// TIA Portal V20 export
// export: Created 2026-04-23T02:21:41.3399534Z, ExportSetting None, DisplayName Totally Integrated Automation Portal, DisplayVersion V20 Update 4, DisplayName TIA Portal Openness, DisplayVersion V20 Update 4, DisplayName TIA Portal Version Control Interface, DisplayVersion V20 Update 4, DisplayName SINAMICS Startdrive Advanced, DisplayVersion V20 SP1 Update 2, DisplayName SINAMICS Startdrive G110M, G120, G120C, G120D, G120P, G115D, DisplayVersion V20 SP1 Update 2, DisplayName SINAMICS Startdrive G130, G150, S120, S150, SINAMICS MV, G220, S200, S210, DisplayVersion V20 SP1 Update 2, DisplayName STEP 7 Professional, DisplayVersion V20 Update 4, DisplayName STEP 7 Safety, DisplayVersion V20 Update 2, DisplayName WinCC Basic/Comfort/Advanced, DisplayVersion V20 Update 4, DisplayName SIMATIC Visualization Architect, DisplayVersion V20 Update 4, DisplayName WinCC Unified, DisplayVersion V20 Update 4, DisplayName SIMATIC Visualization Architect, DisplayVersion V20 Update 4
FUNCTION_BLOCK "LSicar_KistlerPress"   // FB2, LAD
{ S7_Optimized_Access := 'TRUE' }
// stored: MemoryReserve 100, SetENOAutomatically false
   VAR_INPUT
      plantidentifier { ExternalAccessible := 'False'; ExternalVisible := 'False'; ExternalWritable := 'False'} : WString[24];   // Plant/cell identifier string (max 24 chars). Embedded in all ProDiag alarm messages via the @5%s@ placeholder. Set to a unique name per press instance, e.g. KP_ST110_PRS1.
      CarrierID { ExternalAccessible := 'False'; ExternalVisible := 'False'; ExternalWritable := 'False'} : WString[9];   // Carrier or pallet ID (max 9 chars). Passed to the Kistler SmartClient to correlate measurement results with the workpiece carrier for traceability.
      mpSerialNumber { ExternalAccessible := 'False'; ExternalVisible := 'False'; ExternalWritable := 'False'} : String[24];   // Expected workpiece serial number (max 24 chars). Compared against the serial reported by the Kistler device each cycle. A mismatch sets stateAlarm.serialnumbermismatch and blocks sequence start.
      additionaAlarmText { ExternalAccessible := 'False'; ExternalVisible := 'False'; ExternalWritable := 'False'} : WString[15];   // Additional context text (max 15 chars) appended to alarm messages. Use for extra identification, e.g. tool number or station sub-ID.
      tecUnitNumber { ExternalAccessible := 'False'; ExternalVisible := 'False'; ExternalWritable := 'False'} : Int;   // Technical unit number for this press instance. Used for HMI interface routing and identification in multi-press installations.
      enableBlock { ExternalAccessible := 'False'; ExternalVisible := 'False'; ExternalWritable := 'False'} : Bool := TRUE;   // Master block enable. TRUE = block logic active and outputs driven. FALSE = all drive outputs de-energised and alarms suppressed. Default TRUE.
      HardwareOK { ExternalAccessible := 'False'; ExternalVisible := 'False'; ExternalWritable := 'False'} : Bool := TRUE;   // Fieldbus and drive hardware health input. FALSE triggers stateAlarm.hardwareNOK and inhibits all motion commands. Connect to PROFINET device diagnostic or drive ready signal. Default TRUE.
      SafetyOK { ExternalAccessible := 'False'; ExternalVisible := 'False'; ExternalWritable := 'False'} : Bool := TRUE;   // Safety circuit status. FALSE gates all motion commands, de-energises the drive enable, and sets stateAlarm.safetyNOK. Must be TRUE before any press movement is permitted. Default TRUE.
      servoNotInstalled { ExternalAccessible := 'False'; ExternalVisible := 'False'; ExternalWritable := 'False'} : Bool;   // Set TRUE when the servo drive is physically absent (spare station). Bypasses drive-enable and drive-fault alarms and allows the block to run in passthrough mode without a physical axis.
      hardwareID1 { ExternalAccessible := 'False'; ExternalVisible := 'False'; ExternalWritable := 'False'} : HW_IO;   // TIA hardware identifier (HW_IO) for the primary Kistler PROFINET device. Used as LADDR in DPRD_DAT to read the 200-byte cyclic receive telegram each scan.
      hardwareID2 { ExternalAccessible := 'False'; ExternalVisible := 'False'; ExternalWritable := 'False'} : HW_IO;   // TIA hardware identifier (HW_IO) for the secondary Kistler PROFINET device. Used as LADDR in DPWR_DAT to write the transmit telegram to the device.
      smartClientIPAddress { ExternalAccessible := 'False'; ExternalVisible := 'False'; ExternalWritable := 'False'} : String[20];   // IP address string of the Kistler SmartClient application (max 20 chars). Stored for reference and remote configuration. Set to the network address of the Kistler PC running SmartClient.
      mpNumber { ExternalAccessible := 'False'; ExternalVisible := 'False'; ExternalWritable := 'False'} : Byte;   // Measurement program (MP) number to load on the Kistler device. Sent via the fieldbus transmit telegram. Valid range and program definitions are configured on the Kistler SmartClient.
      cfgAdd { ExternalAccessible := 'False'; ExternalVisible := 'False'; ExternalWritable := 'False'} : Byte;   // Starting byte offset in the Kistler fieldbus configuration area. Combined with CfgLentgh to define the read/write window for the configuration data telegram exchange.
      CfgLentgh { ExternalAccessible := 'False'; ExternalVisible := 'False'; ExternalWritable := 'False'} : Byte;   // Length in bytes of the Kistler configuration telegram block. Determines how many bytes are transferred during each configuration read or write operation.
      SelectPageNumber { ExternalAccessible := 'False'; ExternalVisible := 'False'; ExternalWritable := 'False'} : Byte;   // Display page number to activate on the Kistler operator panel or SmartClient HMI. Sent in the transmit telegram each scan.
      selectSequence { ExternalAccessible := 'False'; ExternalVisible := 'False'; ExternalWritable := 'False'} : Byte;   // Sequence profile number to activate on the Kistler device. Sent via the fieldbus transmit telegram to select which measurement sequence to run.
      extStopRequest { ExternalAccessible := 'False'; ExternalVisible := 'False'; ExternalWritable := 'False'} : Bool;   // External stop request from upstream logic (e.g. part-not-present or conveyor fault). Rising edge halts the running sequence gracefully and sets sequenceStopped. Timeout monitored by timeExtStop.
      strobeEnable { ExternalAccessible := 'False'; ExternalVisible := 'False'; ExternalWritable := 'False'} : Bool;   // Gate for the automatic data-strobe pulse. TRUE allows the strobe command to be sent to the Kistler device during a running sequence to trigger data capture.
      startTL { ExternalAccessible := 'False'; ExternalVisible := 'False'; ExternalWritable := 'False'} : Bool;   // Rising edge initiates the teach-learn or reference-position calibration cycle on the Kistler axis. Hold TRUE until the TL cycle is confirmed complete.
      autoRunSequence { ExternalAccessible := 'False'; ExternalVisible := 'False'; ExternalWritable := 'False'} : Bool := FALSE;   // When TRUE the block automatically triggers the measurement sequence on each new cycle trigger. When FALSE the sequence must be started manually via HMI. Default FALSE.
      autoHomePosition { ExternalAccessible := 'False'; ExternalVisible := 'False'; ExternalWritable := 'False'} : Bool;   // When TRUE the axis automatically returns to home position after each sequence completes normally. Disable for processes that require the axis to hold position after pressing.
      autoDriveToReferencePosition { ExternalAccessible := 'False'; ExternalVisible := 'False'; ExternalWritable := 'False'} : Bool;   // When TRUE the axis automatically drives to the reference/calibration position during block initialisation or after a reset. Used for absolute position referencing at startup.
      JogFwd { ExternalAccessible := 'False'; ExternalVisible := 'False'; ExternalWritable := 'False'} : Bool;   // Jog press forward (downward, pressing direction). Drive moves while signal is TRUE. Only active in manual or setup mode. Rate limited by jog speed in parameters.
      JogNeq { ExternalAccessible := 'False'; ExternalVisible := 'False'; ExternalWritable := 'False'} : Bool;   // Jog press negative/backward (upward, retract direction). Drive moves while signal is TRUE. Only active in manual or setup mode.
      continuewait { ExternalAccessible := 'False'; ExternalVisible := 'False'; ExternalWritable := 'False'} : Bool;   // Rising edge clears the waitContinue pause state and resumes sequence execution. Used for operator-confirmation steps in semi-automatic cycles or fault-recovery sequences.
      SequenceEndReset { ExternalAccessible := 'False'; ExternalVisible := 'False'; ExternalWritable := 'False'} : Bool;   // Rising edge resets the Sequenceend, sequenceStopped, and internal sequence-complete flags, clearing the end-of-cycle indication and allowing a new cycle to be triggered.
      enableRunSequence { ExternalAccessible := 'False'; ExternalVisible := 'False'; ExternalWritable := 'False'} : Bool := TRUE;   // Enable gate for sequence execution. FALSE prevents the measurement sequence from starting even if autoRunSequence is TRUE or a manual start is requested. Default TRUE.
      enablehomePos { ExternalAccessible := 'False'; ExternalVisible := 'False'; ExternalWritable := 'False'} : Bool := TRUE;   // Enable gate for home-position return. FALSE prevents the axis from driving to home position even when autoHomePosition is TRUE. Default TRUE.
      externalAlarm { ExternalAccessible := 'False'; ExternalVisible := 'False'; ExternalWritable := 'False'} : Bool;   // External fault injection from another block or interlock. When TRUE, sets stateAlarm.alarm and contributes to GeneralAlarm. Allows upstream faults to be reflected through the Kistler block.
      runWithoutEnable { ExternalAccessible := 'False'; ExternalVisible := 'False'; ExternalWritable := 'False'} : Bool;   // Bypass flag for the opmode enable check. When TRUE the block runs in automatic mode even if the opmode enable signal is not active. Use for commissioning only.
      hideAlarmAll { ExternalAccessible := 'False'; ExternalVisible := 'False'; ExternalWritable := 'False'} : Bool;   // Global alarm suppression. When TRUE all ProDiag alarm messages are suppressed. Does not clear active faults, only prevents message annunciation. Typically driven by a plant-level inhibit.
      hideAlarmMask { ExternalAccessible := 'False'; ExternalVisible := 'False'; ExternalWritable := 'False'} : DWord;   // 32-bit individual alarm suppression mask. Each bit maps to one stateAlarm bit (bit 0 = spare0, bit 1 = hardwareNOK, etc.). Set a bit TRUE to suppress that alarm channel without affecting others.
      OpModeUserInterfaceOut { ExternalAccessible := 'False'; ExternalVisible := 'False'; ExternalWritable := 'False'} : "LSicar_typeOpmodeOut";   // Operating mode data from SYSTEM_DB.OPmode[N].User_Interface_OUT. Contains automaticActive, manualActive, singleStepActive flags and operator preselect requests used to drive mode-selection logic.
      timeOperation { ExternalAccessible := 'False'; ExternalVisible := 'False'; ExternalWritable := 'False'} : Time;   // Maximum allowed duration for a press operation cycle (IEC Time). If the sequence does not complete within this time, stateAlarm.timerMonitorRunSequence is set and the cycle is aborted.
      timeExtStop { ExternalAccessible := 'False'; ExternalVisible := 'False'; ExternalWritable := 'False'} : Time;   // Maximum time allowed for the extStopRequest signal to clear after it rises. If the signal remains TRUE beyond this time, a timeout fault is latched in stateAlarm.
      parameters { ExternalAccessible := 'False'; ExternalVisible := 'False'; ExternalWritable := 'False'} : "LDrive_typeKistlerParameters";   // LDrive_typeKistlerParameters struct. Contains press axis travel limits, force window limits, jog speed, sequence timing parameters, and SmartClient configuration values.
   END_VAR
   VAR_OUTPUT
      GeneralAlarm { ExternalAccessible := 'False'; ExternalVisible := 'False'; ExternalWritable := 'False'} : Bool;   // TRUE when any active unmasked fault condition exists. Drives ProDiag supervision alarm output. Must be FALSE for the ready output to be TRUE.
      AutomaticActive { ExternalAccessible := 'False'; ExternalVisible := 'False'; ExternalWritable := 'False'} : Bool;   // TRUE when the block is operating in automatic mode (opmode automatic active and enableBlock TRUE). Indicates the press is available for production cycles.
      okTotal { ExternalAccessible := 'False'; ExternalVisible := 'False'; ExternalWritable := 'False'} : Bool;   // Pulses TRUE for one scan when the Kistler device reports an OK result for the last completed measurement (all evaluation channels within defined limits).
      nokTotal { ExternalAccessible := 'False'; ExternalVisible := 'False'; ExternalWritable := 'False'} : Bool;   // Pulses TRUE for one scan when the Kistler device reports a NOK result (at least one evaluation channel outside its defined limit window).
      noPass { ExternalAccessible := 'False'; ExternalVisible := 'False'; ExternalWritable := 'False'} : Bool;   // TRUE when the Kistler evaluation reports a no-pass condition for the current measurement program. Distinct from NOK -- indicates an evaluation rule was not met.
      sequenceRunning { ExternalAccessible := 'False'; ExternalVisible := 'False'; ExternalWritable := 'False'} : Bool;   // TRUE while a measurement sequence is actively executing on the press axis. Falls FALSE when the sequence completes, is stopped, or a fault occurs.
      sequenceStopped { ExternalAccessible := 'False'; ExternalVisible := 'False'; ExternalWritable := 'False'} : Bool;   // TRUE after a sequence was interrupted by extStopRequest or a manual stop command. Remains TRUE until cleared by SequenceEndReset rising edge.
      Sequenceend { ExternalAccessible := 'False'; ExternalVisible := 'False'; ExternalWritable := 'False'} : Bool;   // Pulses TRUE for one scan when a sequence completes normally without fault. Cleared by SequenceEndReset rising edge or the start of a new cycle.
      homePos { ExternalAccessible := 'False'; ExternalVisible := 'False'; ExternalWritable := 'False'} : Bool;   // TRUE when the press axis is confirmed at the home/retracted position within the home-position tolerance window defined in parameters.
      referencePos { ExternalAccessible := 'False'; ExternalVisible := 'False'; ExternalWritable := 'False'} : Bool;   // TRUE when the press axis is confirmed at the reference/calibration position. Used to validate absolute position referencing after startup or reset.
      waitContinue { ExternalAccessible := 'False'; ExternalVisible := 'False'; ExternalWritable := 'False'} : Bool;   // TRUE when the block is paused at a wait-for-operator step in the sequence. Cleared by a rising edge on the continuewait input.
      ready { ExternalAccessible := 'False'; ExternalVisible := 'False'; ExternalWritable := 'False'} : Bool;   // TRUE when the block is fault-free, fully enabled, axis at home position, and ready to accept a new cycle trigger. The primary go/no-go signal for upstream sequence control.
      pvCurrentValueX { ExternalAccessible := 'False'; ExternalVisible := 'False'; ExternalWritable := 'False'} : Real;   // Live X-axis process value from the Kistler sensor, typically press position in mm. Scaled from the raw fieldbus data using engineering unit conversion in the Process Values Mapping network.
      pvCurrentValueY { ExternalAccessible := 'False'; ExternalVisible := 'False'; ExternalWritable := 'False'} : Real;   // Live Y-axis process value from the Kistler sensor, typically press force in kN. Scaled from the raw fieldbus data using engineering unit conversion in the Process Values Mapping network.
      pvCurveXminX { ExternalAccessible := 'False'; ExternalVisible := 'False'; ExternalWritable := 'False'} : Real;   // Lower X bound (position) of the active evaluation envelope window. Sourced from the current measurement program parameters on the Kistler device.
      pvCurveXmaxX { ExternalAccessible := 'False'; ExternalVisible := 'False'; ExternalWritable := 'False'} : Real;   // Upper X bound (position) of the active evaluation envelope window. Sourced from the current measurement program parameters on the Kistler device.
      pvCurveYminY { ExternalAccessible := 'False'; ExternalVisible := 'False'; ExternalWritable := 'False'} : Real;   // Lower Y bound (force) of the active evaluation envelope window. Sourced from the current measurement program parameters on the Kistler device.
      pvCurveYmaxY { ExternalAccessible := 'False'; ExternalVisible := 'False'; ExternalWritable := 'False'} : Real;   // Upper Y bound (force) of the active evaluation envelope window. Sourced from the current measurement program parameters on the Kistler device.
      customeProcessValues { ExternalAccessible := 'False'; ExternalVisible := 'False'; ExternalWritable := 'False'} : "LDrive_typeKistlerProcessValues";   // LDrive_typeKistlerProcessValues struct. Full result set from the Kistler evaluation: all channel measured values, individual pass/fail flags, peak force, peak position, and gradient data.
      displayeservoJogSpeed { ExternalAccessible := 'False'; ExternalVisible := 'False'; ExternalWritable := 'False'} : Real;   // Current servo jog speed as a percentage (0-100%). Calculated from the active jog speed parameter and displayed on the HMI for operator awareness during manual axis movement.
      standstill { ExternalAccessible := 'False'; ExternalVisible := 'False'; ExternalWritable := 'False'} : Bool;   // TRUE when the servo axis velocity is confirmed at zero by the drive. Safe condition for clamp operations or position checks that require the press to be stationary.
      MeasurementProgramEcho { ExternalAccessible := 'False'; ExternalVisible := 'False'; ExternalWritable := 'False'} : DInt;   // Echo of the currently active measurement program number confirmed by the Kistler device. Compare against mpNumber input to verify program selection was accepted.
      currentLabel { ExternalAccessible := 'False'; ExternalVisible := 'False'; ExternalWritable := 'False'} : Byte;   // Current sequence step label number as reported by the Kistler device. Indicates which step in the press sequence is active. Used on HMI for step-level diagnostics.
   END_VAR
   VAR_IN_OUT
      interfaceHmi : Array[*] of "LDrive_typeKistlerHmi";
   END_VAR
   VAR
      statDataExchangeReceive { ExternalAccessible := 'False'; ExternalVisible := 'False'; ExternalWritable := 'False'} : "LDrive_typeKistlerPressDataRecv";   // Dynamic array of LDrive_typeKistlerHmi structs, one element per configured press channel. HMI reads status and process values from this array; operator commands and parameter adjustments are written back into it each scan.
      statDataExchangeSend { ExternalAccessible := 'False'; ExternalVisible := 'False'; ExternalWritable := 'False'} : "LDrive_typeKistlerPressDataSend";
      statInstruction { ExternalAccessible := 'False'; ExternalVisible := 'False'; ExternalWritable := 'False'} : Struct
         timeroperation { S7_SetPoint := 'True'} : IEC_TIMER;
         driveEnableTMR { S7_SetPoint := 'True'} : IEC_TIMER;
      END_STRUCT;
      stateAlarm { ExternalAccessible := 'False'; ExternalVisible := 'False'; ExternalWritable := 'False'} : Struct
         spare0 : Bool;
         hardwareNOK : Bool;
         driveenabledNOK : Bool;
         enableRunSequence : Bool;
         enableHomePos : Bool;
         timerMonitorRunSequence : Bool;
         timerMonitorHomePos : Bool;
         timerMonitorReferencePos : Bool;
         noContinueWaitCommand : Bool;
         alarm : Bool;
         spare11 : Bool;
         smesActive : Bool;
         safetyNOK : Bool;
         smst2active : Bool;
         smm1active : Bool;
         serialnumbermismatch : Bool;
         transmissionFault : Bool;
         remoteControlNotActive : Bool;
      END_STRUCT;
      stateHideAlarm { ExternalAccessible := 'False'; ExternalVisible := 'False'; ExternalWritable := 'False'} : Struct
         spare0 : Bool;
         hardwareNOK : Bool;
         transmissionFault : Bool;
         driveEnabledNOK : Bool;
         enableRunSequence : Bool;
         enableHomePos : Bool;
         timerMonitorRunSequence : Bool;
         timerMonitorHomePos : Bool;
         timerMonitorReferencePos : Bool;
         noContinueWaitCommand : Bool;
         Alarm : Bool;
         spare11 : Bool;
         smesactive : Bool;
         safetyNOK : Bool;
         smst2active : Bool;
         smm1Active : Bool;
      END_STRUCT;
      aux { ExternalAccessible := 'False'; ExternalVisible := 'False'; ExternalWritable := 'False'} : Struct
         generalAlarm : Bool := false;
         plantIdentifier : String[24];
         HideAlarmAll : Bool := false;
         manualMode : Bool := false;
         automaticMode : Bool := false;
         singleStepMode : Bool := false;
         setupMode : Bool := false;
         externalAlarm : Bool := false;
         alarmPdNoChange : Bool := false;
         internalAlarmPdNoChange : Bool := false;
         lastAlarmNoPD : UInt := 0;
         lastInternalAlarmNoPD : UInt := 0;
         enableAdvancedCodeView : Bool := false;
         enableReverseCodeView : Bool := false;
         codeViewAdvancedFilter : WString[48];
         codeViewReverseFilter : WString[48];
         iecTimer1 : TON_TIME;
         logicEnable { S7_SetPoint := 'True'} : Bool := false;
         runSequence : Bool := false;
         sequenceEnd : Bool := false;
         dataStrobed : Bool := false;
         SeqEnd : Bool := false;
         remoteControl : Bool := false;
         manualDataStrobe : Bool := false;
         kistlerDataDB : Int := 0;
         pulse : Array[0..16] of Bool;
         Interface : DWord;
      END_STRUCT;
      ons { ExternalAccessible := 'False'; ExternalVisible := 'False'; ExternalWritable := 'False'} : Array[0..16] of Bool;
      statTimeExpire { ExternalAccessible := 'False'; ExternalVisible := 'False'; ExternalWritable := 'False'} : Struct
         operating : Bool;
         position_pLeft : Bool;
         selaypair_mon : Bool;
         dwellTimeWork : Bool;
         dwellTimeHome : Bool;
      END_STRUCT;
      statAlarmtextHeader { ExternalAccessible := 'False'; ExternalVisible := 'False'; ExternalWritable := 'False'} : WString[60];
      statAlarmtextFooter { ExternalAccessible := 'False'; ExternalVisible := 'False'; ExternalWritable := 'False'} : WString[24];
      statPalletID { ExternalAccessible := 'False'; ExternalVisible := 'False'; ExternalWritable := 'False'} : WString[9];
      statAlarmNoPD { ExternalAccessible := 'False'; ExternalVisible := 'False'; ExternalWritable := 'False'} : UInt;
      statInternalAlarmNoPD { ExternalAccessible := 'False'; ExternalVisible := 'False'; ExternalWritable := 'False'} : UInt;
      statHideAlarmMessagesPD { ExternalAccessible := 'False'; ExternalVisible := 'False'; ExternalWritable := 'False'} : Bool;
      statGlobalTecunitWarningTestListItem { ExternalAccessible := 'False'; ExternalVisible := 'False'; ExternalWritable := 'False'} : USInt := 92;
      statCodeViewAdvanceCond { ExternalAccessible := 'False'; ExternalVisible := 'False'; ExternalWritable := 'False'} : TON_TIME;
      statCodeViewReverseCond { ExternalAccessible := 'False'; ExternalVisible := 'False'; ExternalWritable := 'False'; S7_SetPoint := 'True'} : TON_TIME;
      statdriveDelayTimer { ExternalAccessible := 'False'; ExternalVisible := 'False'; ExternalWritable := 'False'; S7_SetPoint := 'True'} : TON_TIME;
      tof { ExternalAccessible := 'False'; ExternalVisible := 'False'; ExternalWritable := 'False'; S7_SetPoint := 'True'} : TON_TIME;
      statSerialByteIndex { ExternalAccessible := 'False'; ExternalVisible := 'False'; ExternalWritable := 'False'; S7_SetPoint := 'True'} : Int;
      statAlarmByteIndex { ExternalAccessible := 'False'; ExternalVisible := 'False'; ExternalWritable := 'False'} : Int;
      statStringIndex { ExternalAccessible := 'False'; ExternalVisible := 'False'; ExternalWritable := 'False'} : Int;
      statSerialOutput { ExternalAccessible := 'False'; ExternalVisible := 'False'; ExternalWritable := 'False'} : String[24];
      instKistlerOnDelay { ExternalAccessible := 'False'; ExternalVisible := 'False'; ExternalWritable := 'False'} : TON_TIME;
      internalFaultCode { ExternalAccessible := 'False'; ExternalVisible := 'False'; ExternalWritable := 'False'; S7_SetPoint := 'True'} : Array[0..63] of Bool;
      AlarmTextConstants { ExternalAccessible := 'False'; ExternalVisible := 'False'; ExternalWritable := 'False'} : Array[0..63] of Int;
      i { ExternalAccessible := 'False'; ExternalVisible := 'False'; ExternalWritable := 'False'} : Int;
   END_VAR
   VAR_TEMP
      tempReturnValueRead : Int;
      tempReturnValueWrite : Int;
      tempMPEcho : SInt;
      tempReadOK : Bool;
      tempWriteOK : Bool;
      tempValue : DWord;
      tempString : String[24];
      tempSerialLength : USInt;
      tempIndex : USInt;
      tempDword : DWord;
      tempErrorValue : Int;
      tempDint : DInt;
   END_VAR
   VAR CONSTANT
      cfgKistlerOnDelay : Time := T#1s;
   END_VAR
   VAR_TEMP   // added for the SCL form of the ladder/FBD networks
      _w1 : Bool;
      _w2 : Bool;
      _w3 : Bool;
      _w4 : Bool;
      _w5 : Bool;
      _w6 : Bool;
      _w7 : Bool;
   END_VAR
BEGIN

REGION Network 1 (SCL): Block Header
   // ================================================================================
   //   LSicar_KistlerPress  --  Kistler Force/Press Monitor Interface Block
   // ================================================================================
   // 
   // DESCRIPTION
   //   Standardised interface block for Kistler press-force monitoring systems
   //   connected via PROFINET IO. Manages the full press cycle: drive enabling,
   //   measurement program selection, sequence execution, force/position data
   //   extraction, result evaluation, and alarm annunciation.
   // 
   //   Communicates with the Kistler device using DPRD_DAT / DPWR_DAT over two
   //   PROFINET hardware identifiers (hardwareID1/hardwareID2) exchanging a
   //   200-byte cyclic telegram each scan.
   // 
   // FEATURES
   //   - Fieldbus I/O       : DPRD_DAT / DPWR_DAT cyclic 200-byte telegram exchange
   //   - Drive control      : Enable, jog forward/backward, home, reference position
   //   - Measurement        : MP selection, sequence start/stop, strobe, result capture
   //   - Result outputs     : OK/NOK/NoPass flags, X/Y process values, envelope bounds
   //   - Serial validation  : Workpiece serial number check before sequence start
   //   - Alarm management   : 18-bit stateAlarm struct, per-bit mask, global suppress
   //   - HMI interface      : Dynamic LDrive_typeKistlerHmi array for operator panel
   //   - Timeout monitoring : Operation cycle timer, ext-stop timeout
   // 
   // INTERFACE SUMMARY
   //   Input  : plantidentifier, CarrierID, mpSerialNumber, additionaAlarmText,
   //            tecUnitNumber, enableBlock, HardwareOK, SafetyOK, servoNotInstalled,
   //            hardwareID1, hardwareID2, smartClientIPAddress, mpNumber, cfgAdd,
   //            CfgLentgh, SelectPageNumber, selectSequence, extStopRequest,
   //            strobeEnable, startTL, autoRunSequence, autoHomePosition,
   //            autoDriveToReferencePosition, JogFwd, JogNeq, continuewait,
   //            SequenceEndReset, enableRunSequence, enablehomePos, externalAlarm,
   //            runWithoutEnable, hideAlarmAll, hideAlarmMask,
   //            OpModeUserInterfaceOut, timeOperation, timeExtStop, parameters
   //   InOut  : interfaceHmi (dynamic array of LDrive_typeKistlerHmi)
   //   Output : GeneralAlarm, AutomaticActive, okTotal, nokTotal, noPass,
   //            sequenceRunning, sequenceStopped, Sequenceend, homePos,
   //            referencePos, waitContinue, ready, pvCurrentValueX, pvCurrentValueY,
   //            pvCurveXminX, pvCurveXmaxX, pvCurveYminY, pvCurveYmaxY,
   //            customeProcessValues, displayeservoJogSpeed, standstill,
   //            MeasurementProgramEcho, currentLabel
   // 
   // NETWORK LAYOUT
   //   Net  1  Block Header -- documentation only (this network)
   //   Net  2  Read RAW Data from Kistler (SCL - DPRD_DAT)
   //   Net  3  Read OK -- DPRD_DAT error check
   //   Net  4  External Alarm
   //   Net  5  Set Hide Alarm -- mask mapping
   //   Net  6  Hide Alarm -- suppression logic
   //   Net  7  Mode Selection
   //   Net  8  Clear Faults
   //   Net  9  Enable the Drive
   //   Net 10  Control Remotely
   //   Net 11  Turn to Auto mode remotely
   //   Net 12  SetupMP and Pages
   //   Net 13  DataStrobe Manually
   //   Net 14  DataStrobe Acknowledged
   //   Net 15  Strobe data
   //   Net 16  Sequence End (detect)
   //   Net 17  Run the sequence
   //   Net 18  Validate Serial Before Running
   //   Net 19  Run Sequence (state)
   //   Net 20  Initiate TL Devices
   //   Net 21  Monitor Operation Timeouts
   //   Net 22  Select Sequence
   //   Net 23  SeqExtStopReq
   //   Net 24  Resume After Error
   //   Net 25  Sequence End (latch)
   //   Net 26  Flag Internal Seq End Flags
   //   Net 27  ReturnHomePos
   //   Net 28  DrivetoRefPos
   //   Net 29  JOG Forward
   //   Net 30  JOG Backward
   //   Net 31  Map Incoming Field Bus data (200 bytes)
   //   Net 32  Map Digital Signals
   //   Net 33  Write Raw Data to Kistler (DPWR_DAT)
   //   Net 34  Write OK -- DPWR_DAT error check
   //   Net 35  Display Seq END
   //   Net 36  Map Fixed Fieldbus outputs
   //   Net 37  Process Values Mapping
   //   Net 38  Alarms
   //   Net 39  Evaluate Internal Alarms
   //   Net 40  Fault General Alarm
   //   Net 41  Map Alarms to HMI Interface
   // 
   // VERSION HISTORY
   //   0.0.1  Initial release.
   //   0.0.2  Added block-header documentation network, interface member comments,
   //          and network comments on all 40 networks.
   // 
   // AUTHOR  : Amperesand
   // COMPANY : Amperesand Pte. Ltd.
   // LICENSE : Internal use only -- Amperesand Engineering
   // ================================================================================
   REGION Block Header
   END_REGION
END_REGION

REGION Network 2 (SCL): Read RAW Data from Kistler
   // DPRD_DAT reads the 200-byte cyclic receive telegram from the primary Kistler PROFINET device (hardwareID1) into statDataExchangeReceive. Return value stored in tempReturnValueRead for error checking in the next network.
       #tempReturnValueRead := DPRD_DAT(LADDR := #hardwareID1, RECORD => #statDataExchangeReceive);    // Read from Kistler
END_REGION

REGION Network 3: Read OK
   // Evaluates the DPRD_DAT return value. A non-zero value indicates a fieldbus communication fault; sets stateAlarm.transmissionFault to trigger the transmission fault alarm.
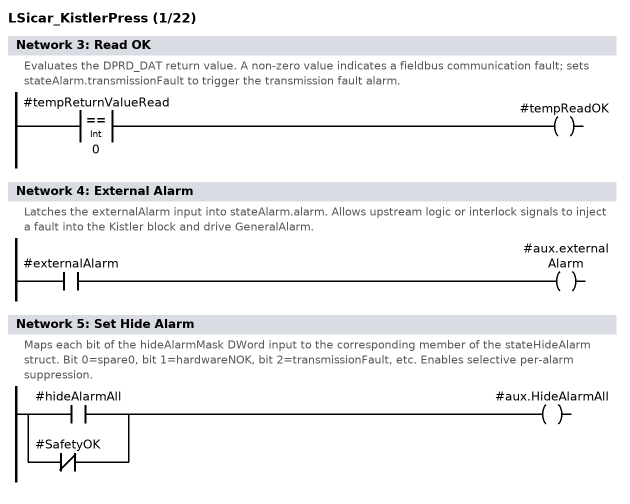
   RUNG wire#powerrail
      { S7_Templates := "SrcType := Int" } EQ_Contact(in1 := #tempReturnValueRead, in2 := 0)
      Coil( #tempReadOK )
   END_RUNG
   // the same network as SCL:
   #tempReadOK := #tempReturnValueRead = 0;
END_REGION

REGION Network 4: External Alarm
   // Latches the externalAlarm input into stateAlarm.alarm. Allows upstream logic or interlock signals to inject a fault into the Kistler block and drive GeneralAlarm.
   RUNG wire#powerrail
      Contact( #externalAlarm )
      Coil( #aux.externalAlarm )
   END_RUNG
   // the same network as SCL:
   #aux.externalAlarm := #externalAlarm;
END_REGION

REGION Network 5: Set Hide Alarm
   // Maps each bit of the hideAlarmMask DWord input to the corresponding member of the stateHideAlarm struct. Bit 0=spare0, bit 1=hardwareNOK, bit 2=transmissionFault, etc. Enables selective per-alarm suppression.
   RUNG wire#powerrail
      Contact( #hideAlarmAll )
      wire#w1
      Coil( #aux.HideAlarmAll )
   END_RUNG
   RUNG wire#powerrail
      I_Contact( #SafetyOK )
   END_RUNG wire#w1
   // the same network as SCL:
   #aux.HideAlarmAll := #hideAlarmAll OR NOT #SafetyOK;
END_REGION

REGION Network 6: Hide Alarm
   // Applies alarm suppression logic. Each stateAlarm bit is ANDed with its stateHideAlarm counterpart (after applying hideAlarmAll). Result drives the active alarm state used in Fault General Alarm network.
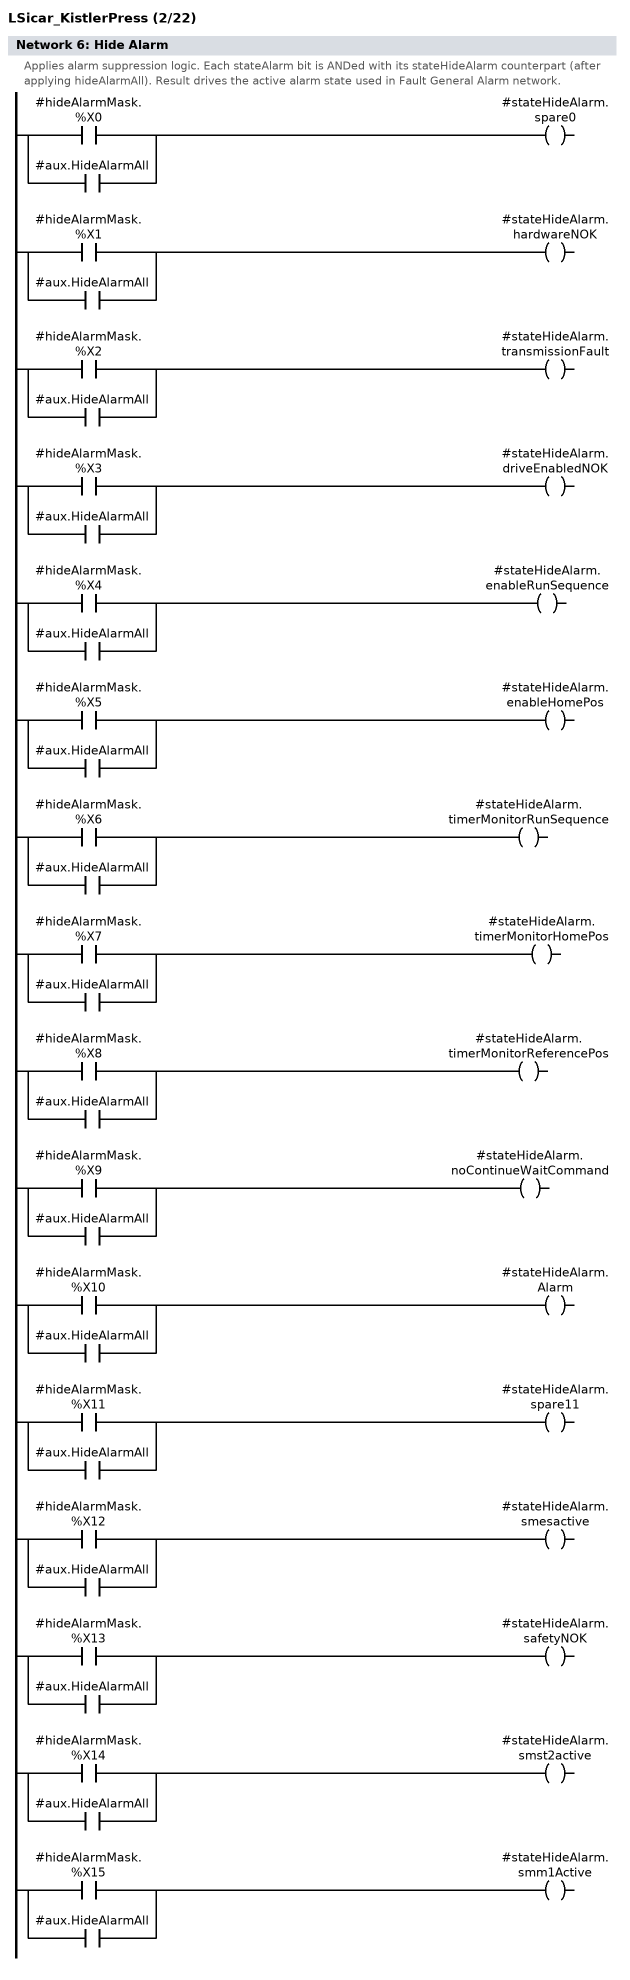
   RUNG wire#powerrail
      Contact( #hideAlarmMask.%X0 )
      wire#w1
      Coil( #stateHideAlarm.spare0 )
   END_RUNG
   RUNG wire#powerrail
      Contact( #aux.HideAlarmAll )
   END_RUNG wire#w1
   RUNG wire#powerrail
      Contact( #hideAlarmMask.%X1 )
      wire#w2
      Coil( #stateHideAlarm.hardwareNOK )
   END_RUNG
   RUNG wire#powerrail
      Contact( #aux.HideAlarmAll )
   END_RUNG wire#w2
   RUNG wire#powerrail
      Contact( #hideAlarmMask.%X2 )
      wire#w3
      Coil( #stateHideAlarm.transmissionFault )
   END_RUNG
   RUNG wire#powerrail
      Contact( #aux.HideAlarmAll )
   END_RUNG wire#w3
   RUNG wire#powerrail
      Contact( #hideAlarmMask.%X3 )
      wire#w4
      Coil( #stateHideAlarm.driveEnabledNOK )
   END_RUNG
   RUNG wire#powerrail
      Contact( #aux.HideAlarmAll )
   END_RUNG wire#w4
   RUNG wire#powerrail
      Contact( #hideAlarmMask.%X4 )
      wire#w5
      Coil( #stateHideAlarm.enableRunSequence )
   END_RUNG
   RUNG wire#powerrail
      Contact( #aux.HideAlarmAll )
   END_RUNG wire#w5
   RUNG wire#powerrail
      Contact( #hideAlarmMask.%X5 )
      wire#w6
      Coil( #stateHideAlarm.enableHomePos )
   END_RUNG
   RUNG wire#powerrail
      Contact( #aux.HideAlarmAll )
   END_RUNG wire#w6
   RUNG wire#powerrail
      Contact( #hideAlarmMask.%X6 )
      wire#w7
      Coil( #stateHideAlarm.timerMonitorRunSequence )
   END_RUNG
   RUNG wire#powerrail
      Contact( #aux.HideAlarmAll )
   END_RUNG wire#w7
   RUNG wire#powerrail
      Contact( #hideAlarmMask.%X7 )
      wire#w8
      Coil( #stateHideAlarm.timerMonitorHomePos )
   END_RUNG
   RUNG wire#powerrail
      Contact( #aux.HideAlarmAll )
   END_RUNG wire#w8
   RUNG wire#powerrail
      Contact( #hideAlarmMask.%X8 )
      wire#w9
      Coil( #stateHideAlarm.timerMonitorReferencePos )
   END_RUNG
   RUNG wire#powerrail
      Contact( #aux.HideAlarmAll )
   END_RUNG wire#w9
   RUNG wire#powerrail
      Contact( #hideAlarmMask.%X9 )
      wire#w10
      Coil( #stateHideAlarm.noContinueWaitCommand )
   END_RUNG
   RUNG wire#powerrail
      Contact( #aux.HideAlarmAll )
   END_RUNG wire#w10
   RUNG wire#powerrail
      Contact( #hideAlarmMask.%X10 )
      wire#w11
      Coil( #stateHideAlarm.Alarm )
   END_RUNG
   RUNG wire#powerrail
      Contact( #aux.HideAlarmAll )
   END_RUNG wire#w11
   RUNG wire#powerrail
      Contact( #hideAlarmMask.%X11 )
      wire#w12
      Coil( #stateHideAlarm.spare11 )
   END_RUNG
   RUNG wire#powerrail
      Contact( #aux.HideAlarmAll )
   END_RUNG wire#w12
   RUNG wire#powerrail
      Contact( #hideAlarmMask.%X12 )
      wire#w13
      Coil( #stateHideAlarm.smesactive )
   END_RUNG
   RUNG wire#powerrail
      Contact( #aux.HideAlarmAll )
   END_RUNG wire#w13
   RUNG wire#powerrail
      Contact( #hideAlarmMask.%X13 )
      wire#w14
      Coil( #stateHideAlarm.safetyNOK )
   END_RUNG
   RUNG wire#powerrail
      Contact( #aux.HideAlarmAll )
   END_RUNG wire#w14
   RUNG wire#powerrail
      Contact( #hideAlarmMask.%X14 )
      wire#w15
      Coil( #stateHideAlarm.smst2active )
   END_RUNG
   RUNG wire#powerrail
      Contact( #aux.HideAlarmAll )
   END_RUNG wire#w15
   RUNG wire#powerrail
      Contact( #hideAlarmMask.%X15 )
      wire#w16
      Coil( #stateHideAlarm.smm1Active )
   END_RUNG
   RUNG wire#powerrail
      Contact( #aux.HideAlarmAll )
   END_RUNG wire#w16
   // the same network as SCL:
   #stateHideAlarm.spare0 := #hideAlarmMask.%X0 OR #aux.HideAlarmAll;
   #stateHideAlarm.hardwareNOK := #hideAlarmMask.%X1 OR #aux.HideAlarmAll;
   #stateHideAlarm.transmissionFault := #hideAlarmMask.%X2 OR #aux.HideAlarmAll;
   #stateHideAlarm.driveEnabledNOK := #hideAlarmMask.%X3 OR #aux.HideAlarmAll;
   #stateHideAlarm.enableRunSequence := #hideAlarmMask.%X4 OR #aux.HideAlarmAll;
   #stateHideAlarm.enableHomePos := #hideAlarmMask.%X5 OR #aux.HideAlarmAll;
   #stateHideAlarm.timerMonitorRunSequence := #hideAlarmMask.%X6 OR #aux.HideAlarmAll;
   #stateHideAlarm.timerMonitorHomePos := #hideAlarmMask.%X7 OR #aux.HideAlarmAll;
   #stateHideAlarm.timerMonitorReferencePos := #hideAlarmMask.%X8 OR #aux.HideAlarmAll;
   #stateHideAlarm.noContinueWaitCommand := #hideAlarmMask.%X9 OR #aux.HideAlarmAll;
   #stateHideAlarm.Alarm := #hideAlarmMask.%X10 OR #aux.HideAlarmAll;
   #stateHideAlarm.spare11 := #hideAlarmMask.%X11 OR #aux.HideAlarmAll;
   #stateHideAlarm.smesactive := #hideAlarmMask.%X12 OR #aux.HideAlarmAll;
   #stateHideAlarm.safetyNOK := #hideAlarmMask.%X13 OR #aux.HideAlarmAll;
   #stateHideAlarm.smst2active := #hideAlarmMask.%X14 OR #aux.HideAlarmAll;
   #stateHideAlarm.smm1Active := #hideAlarmMask.%X15 OR #aux.HideAlarmAll;
END_REGION

REGION Network 7: Mode Selection
   // Reads OpModeUserInterfaceOut and maps automaticActive, manualActive, singleStepActive, and setup mode flags into aux state variables. These aux flags gate downstream sequence and drive control networks.
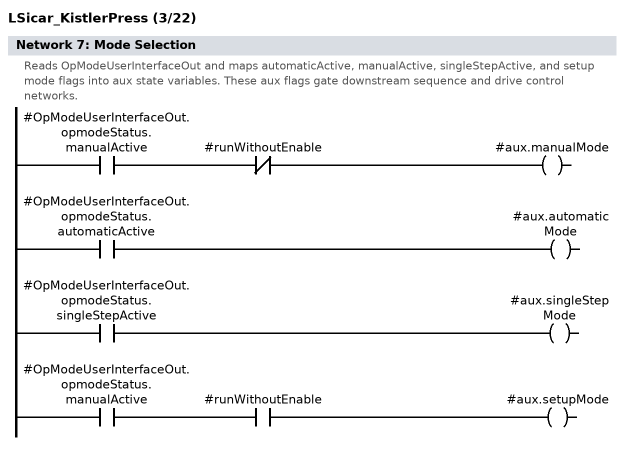
   RUNG wire#powerrail
      Contact( #OpModeUserInterfaceOut.opmodeStatus.manualActive )
      I_Contact( #runWithoutEnable )
      Coil( #aux.manualMode )
   END_RUNG
   RUNG wire#powerrail
      Contact( #OpModeUserInterfaceOut.opmodeStatus.automaticActive )
      Coil( #aux.automaticMode )
   END_RUNG
   RUNG wire#powerrail
      Contact( #OpModeUserInterfaceOut.opmodeStatus.singleStepActive )
      Coil( #aux.singleStepMode )
   END_RUNG
   RUNG wire#powerrail
      Contact( #OpModeUserInterfaceOut.opmodeStatus.manualActive )
      Contact( #runWithoutEnable )
      Coil( #aux.setupMode )
   END_RUNG
   // the same network as SCL:
   #aux.manualMode := #OpModeUserInterfaceOut.opmodeStatus.manualActive AND NOT #runWithoutEnable;
   #aux.automaticMode := #OpModeUserInterfaceOut.opmodeStatus.automaticActive;
   #aux.singleStepMode := #OpModeUserInterfaceOut.opmodeStatus.singleStepActive;
   #aux.setupMode := #OpModeUserInterfaceOut.opmodeStatus.manualActive AND #runWithoutEnable;
END_REGION

REGION Network 8: Clear Faults
   // On a rising edge reset command from HMI or SequenceEndReset, clears all latched stateAlarm fault bits except hardware and safety faults. Resets GeneralAlarm provided no active hardware/safety faults remain.
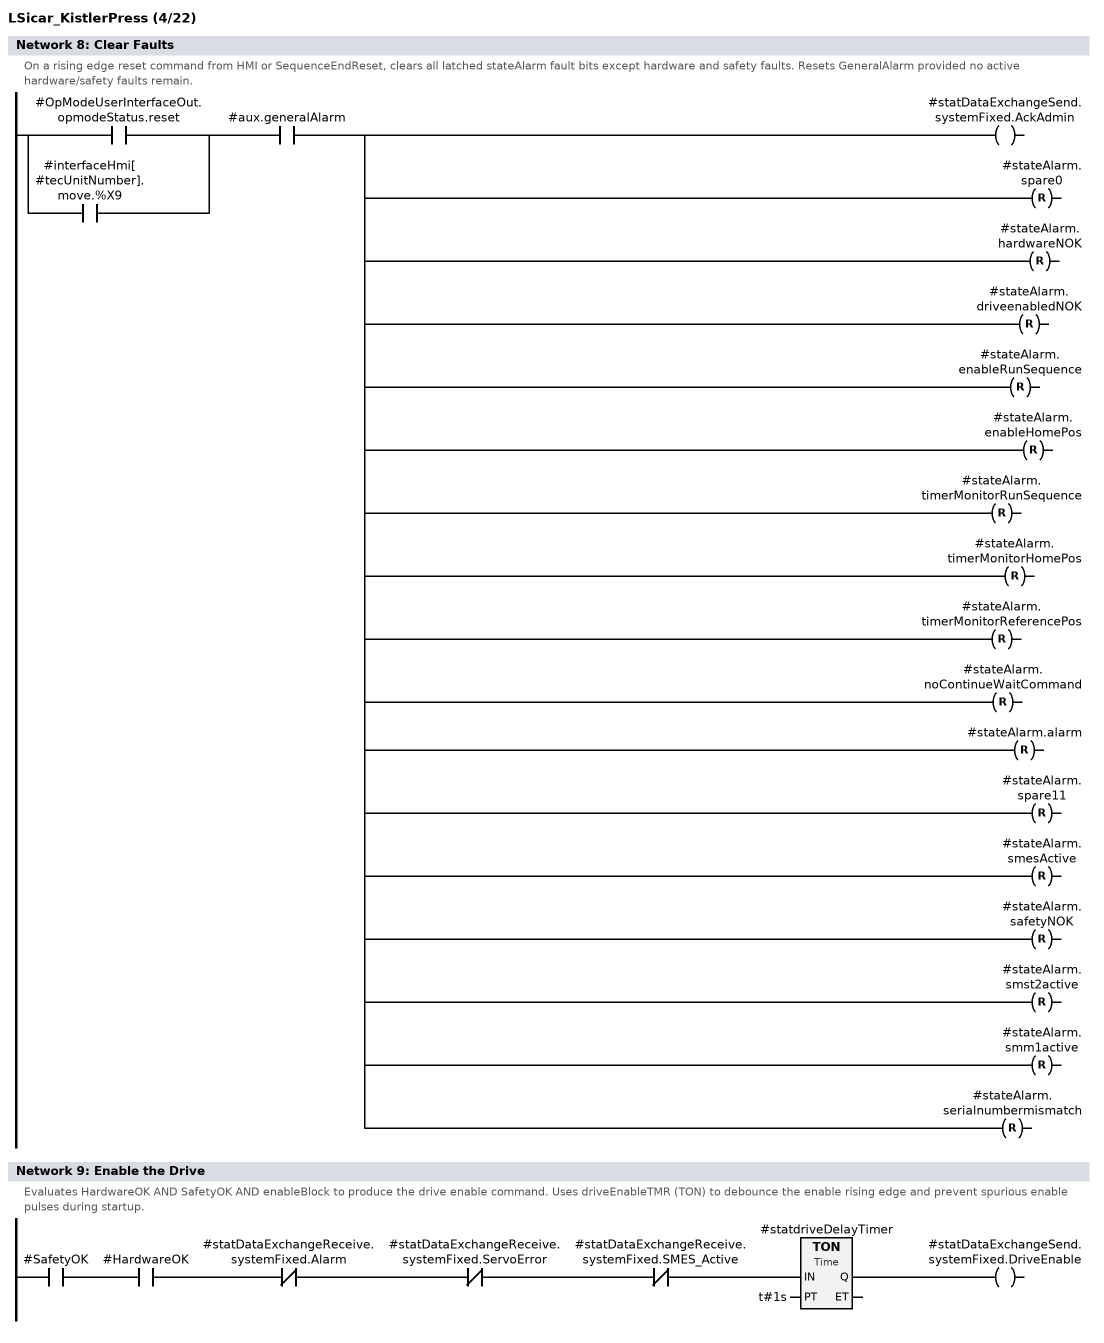
   RUNG wire#powerrail
      Contact( #OpModeUserInterfaceOut.opmodeStatus.reset )
      wire#w1
      Contact( #aux.generalAlarm )
      wire#w2
      Coil( #statDataExchangeSend.systemFixed.AckAdmin )
   END_RUNG
   RUNG wire#powerrail
      Contact( #interfaceHmi[#tecUnitNumber].move.%X9 )
   END_RUNG wire#w1
   RUNG wire#w2
      R_Coil( #stateAlarm.spare0 )
   END_RUNG
   RUNG wire#w2
      R_Coil( #stateAlarm.hardwareNOK )
   END_RUNG
   RUNG wire#w2
      R_Coil( #stateAlarm.driveenabledNOK )
   END_RUNG
   RUNG wire#w2
      R_Coil( #stateAlarm.enableRunSequence )
   END_RUNG
   RUNG wire#w2
      R_Coil( #stateAlarm.enableHomePos )
   END_RUNG
   RUNG wire#w2
      R_Coil( #stateAlarm.timerMonitorRunSequence )
   END_RUNG
   RUNG wire#w2
      R_Coil( #stateAlarm.timerMonitorHomePos )
   END_RUNG
   RUNG wire#w2
      R_Coil( #stateAlarm.timerMonitorReferencePos )
   END_RUNG
   RUNG wire#w2
      R_Coil( #stateAlarm.noContinueWaitCommand )
   END_RUNG
   RUNG wire#w2
      R_Coil( #stateAlarm.alarm )
   END_RUNG
   RUNG wire#w2
      R_Coil( #stateAlarm.spare11 )
   END_RUNG
   RUNG wire#w2
      R_Coil( #stateAlarm.smesActive )
   END_RUNG
   RUNG wire#w2
      R_Coil( #stateAlarm.safetyNOK )
   END_RUNG
   RUNG wire#w2
      R_Coil( #stateAlarm.smst2active )
   END_RUNG
   RUNG wire#w2
      R_Coil( #stateAlarm.smm1active )
   END_RUNG
   RUNG wire#w2
      R_Coil( #stateAlarm.serialnumbermismatch )
   END_RUNG
   // the same network as SCL:
   #statDataExchangeSend.systemFixed.AckAdmin := (#OpModeUserInterfaceOut.opmodeStatus.reset OR #interfaceHmi[#tecUnitNumber].move.%X9) AND #aux.generalAlarm;
   IF #statDataExchangeSend.systemFixed.AckAdmin THEN
       #stateAlarm.spare0 := FALSE;
       #stateAlarm.hardwareNOK := FALSE;
       #stateAlarm.driveenabledNOK := FALSE;
       #stateAlarm.enableRunSequence := FALSE;
       #stateAlarm.enableHomePos := FALSE;
       #stateAlarm.timerMonitorRunSequence := FALSE;
       #stateAlarm.timerMonitorHomePos := FALSE;
       #stateAlarm.timerMonitorReferencePos := FALSE;
       #stateAlarm.noContinueWaitCommand := FALSE;
       #stateAlarm.alarm := FALSE;
       #stateAlarm.spare11 := FALSE;
       #stateAlarm.smesActive := FALSE;
       #stateAlarm.safetyNOK := FALSE;
       #stateAlarm.smst2active := FALSE;
       #stateAlarm.smm1active := FALSE;
       #stateAlarm.serialnumbermismatch := FALSE;
   END_IF;
END_REGION

REGION Network 9: Enable the Drive
   // Evaluates HardwareOK AND SafetyOK AND enableBlock to produce the drive enable command. Uses driveEnableTMR (TON) to debounce the enable rising edge and prevent spurious enable pulses during startup.
   RUNG wire#powerrail
      Contact( #SafetyOK )
      Contact( #HardwareOK )
      I_Contact( #statDataExchangeReceive.systemFixed.Alarm )
      I_Contact( #statDataExchangeReceive.systemFixed.ServoError )
      I_Contact( #statDataExchangeReceive.systemFixed.SMES_Active )
      { S7_Templates := "time_type := Time" } #statdriveDelayTimer.TON(pt := t#1s, et =>)
      Coil( #statDataExchangeSend.systemFixed.DriveEnable )
   END_RUNG
   // the same network as SCL:
   #statdriveDelayTimer(IN := #SafetyOK AND #HardwareOK AND NOT #statDataExchangeReceive.systemFixed.Alarm AND NOT #statDataExchangeReceive.systemFixed.ServoError AND NOT #statDataExchangeReceive.systemFixed.SMES_Active,   // TON
                        PT := t#1s);
   #statDataExchangeSend.systemFixed.DriveEnable := #statdriveDelayTimer.Q;
END_REGION

REGION Network 10: Control Remotely
   // Sets aux.remoteControl TRUE when the Kistler SmartClient is connected and active, as indicated by the remote-control status flag in statDataExchangeReceive. Enables SmartClient to override local control.
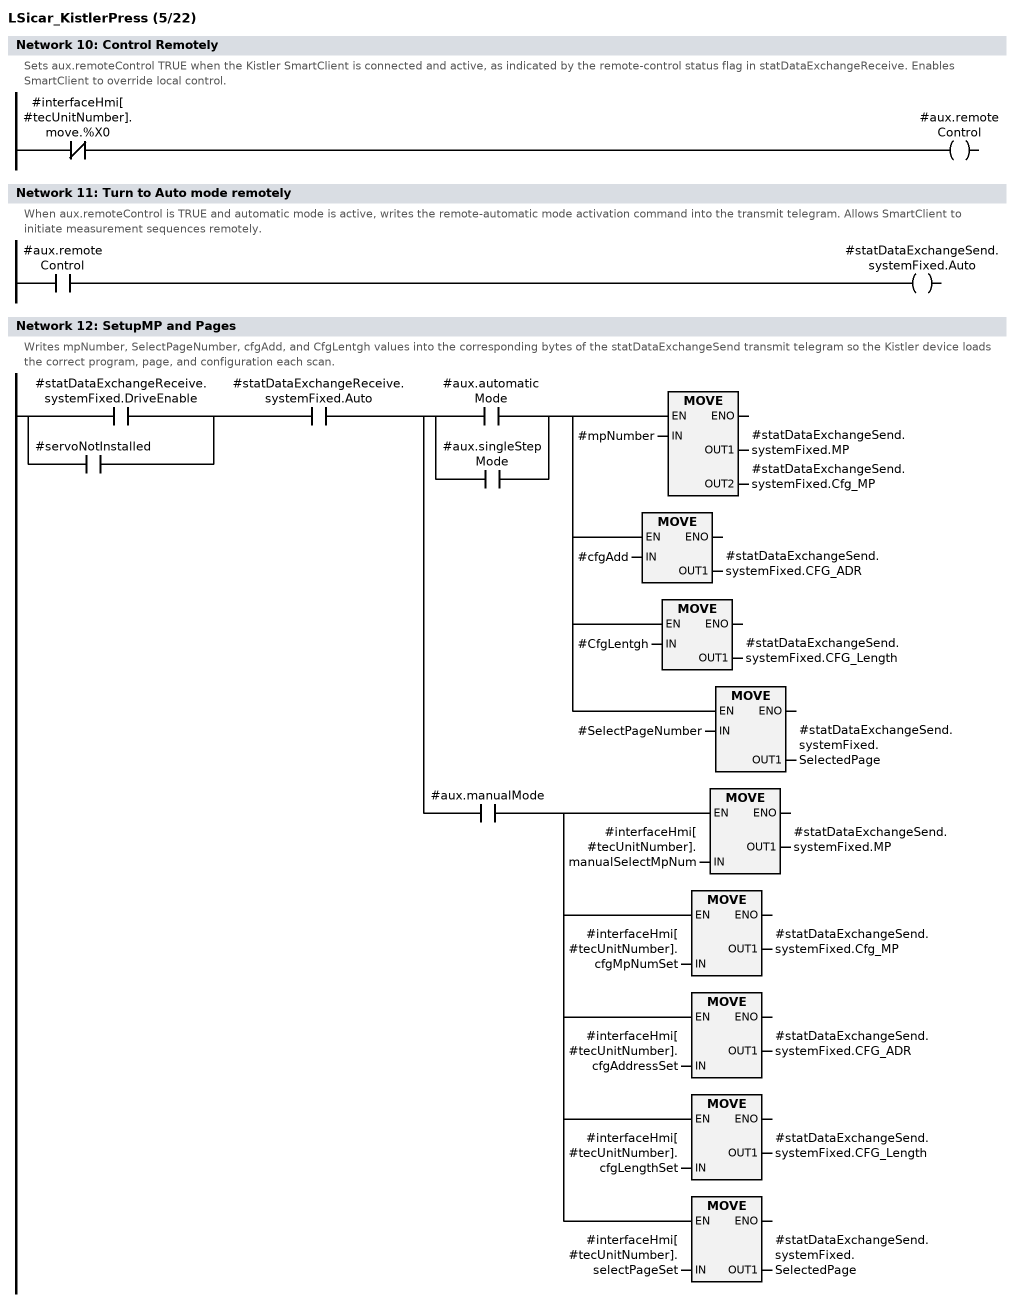
   RUNG wire#powerrail
      I_Contact( #interfaceHmi[#tecUnitNumber].move.%X0 )
      Coil( #aux.remoteControl )
   END_RUNG
   // the same network as SCL:
   #aux.remoteControl := NOT #interfaceHmi[#tecUnitNumber].move.%X0;
END_REGION

REGION Network 11: Turn to Auto mode remotely
   // When aux.remoteControl is TRUE and automatic mode is active, writes the remote-automatic mode activation command into the transmit telegram. Allows SmartClient to initiate measurement sequences remotely.
   RUNG wire#powerrail
      Contact( #aux.remoteControl )
      Coil( #statDataExchangeSend.systemFixed.Auto )
   END_RUNG
   // the same network as SCL:
   #statDataExchangeSend.systemFixed.Auto := #aux.remoteControl;
END_REGION

REGION Network 12: SetupMP and Pages
   // Writes mpNumber, SelectPageNumber, cfgAdd, and CfgLentgh values into the corresponding bytes of the statDataExchangeSend transmit telegram so the Kistler device loads the correct program, page, and configuration each scan.
   RUNG wire#powerrail
      Contact( #statDataExchangeReceive.systemFixed.DriveEnable )
      wire#w1
      Contact( #statDataExchangeReceive.systemFixed.Auto )
      wire#w2
      Contact( #aux.automaticMode )
      wire#w3
      Move(in := #mpNumber, out1 => #statDataExchangeSend.systemFixed.MP, out2 => #statDataExchangeSend.systemFixed.Cfg_MP)
   END_RUNG
   RUNG wire#powerrail
      Contact( #servoNotInstalled )
   END_RUNG wire#w1
   RUNG wire#w2
      Contact( #aux.singleStepMode )
   END_RUNG wire#w3
   RUNG wire#w3
      Move(in := #cfgAdd, out1 => #statDataExchangeSend.systemFixed.CFG_ADR)
   END_RUNG
   RUNG wire#w3
      Move(in := #CfgLentgh, out1 => #statDataExchangeSend.systemFixed.CFG_Length)
   END_RUNG
   RUNG wire#w3
      Move(in := #SelectPageNumber, out1 => #statDataExchangeSend.systemFixed.SelectedPage)
   END_RUNG
   RUNG wire#w2
      Contact( #aux.manualMode )
      wire#w4
      Move(in := #interfaceHmi[#tecUnitNumber].manualSelectMpNum, out1 => #statDataExchangeSend.systemFixed.MP)
   END_RUNG
   RUNG wire#w4
      Move(in := #interfaceHmi[#tecUnitNumber].cfgMpNumSet, out1 => #statDataExchangeSend.systemFixed.Cfg_MP)
   END_RUNG
   RUNG wire#w4
      Move(in := #interfaceHmi[#tecUnitNumber].cfgAddressSet, out1 => #statDataExchangeSend.systemFixed.CFG_ADR)
   END_RUNG
   RUNG wire#w4
      Move(in := #interfaceHmi[#tecUnitNumber].cfgLengthSet, out1 => #statDataExchangeSend.systemFixed.CFG_Length)
   END_RUNG
   RUNG wire#w4
      Move(in := #interfaceHmi[#tecUnitNumber].selectPageSet, out1 => #statDataExchangeSend.systemFixed.SelectedPage)
   END_RUNG
   // the same network as SCL:
   #_w1 := (#statDataExchangeReceive.systemFixed.DriveEnable OR #servoNotInstalled) AND #statDataExchangeReceive.systemFixed.Auto;
   IF #_w1 AND (#aux.automaticMode OR #aux.singleStepMode) THEN
       #statDataExchangeSend.systemFixed.MP := #mpNumber;
       #statDataExchangeSend.systemFixed.Cfg_MP := #mpNumber;
       #statDataExchangeSend.systemFixed.CFG_ADR := #cfgAdd;
       #statDataExchangeSend.systemFixed.CFG_Length := #CfgLentgh;
       #statDataExchangeSend.systemFixed.SelectedPage := #SelectPageNumber;
   END_IF;
   IF #_w1 AND #aux.manualMode THEN
       #statDataExchangeSend.systemFixed.MP := #interfaceHmi[#tecUnitNumber].manualSelectMpNum;
       #statDataExchangeSend.systemFixed.Cfg_MP := #interfaceHmi[#tecUnitNumber].cfgMpNumSet;
       #statDataExchangeSend.systemFixed.CFG_ADR := #interfaceHmi[#tecUnitNumber].cfgAddressSet;
       #statDataExchangeSend.systemFixed.CFG_Length := #interfaceHmi[#tecUnitNumber].cfgLengthSet;
       #statDataExchangeSend.systemFixed.SelectedPage := #interfaceHmi[#tecUnitNumber].selectPageSet;
   END_IF;
END_REGION

REGION Network 13: DataStrobe Manually
   // Handles manual data strobe triggered from the HMI (aux.manualDataStrobe). Generates a one-scan strobe pulse in the transmit telegram to trigger a manual data capture on the Kistler device for test or debug purposes.
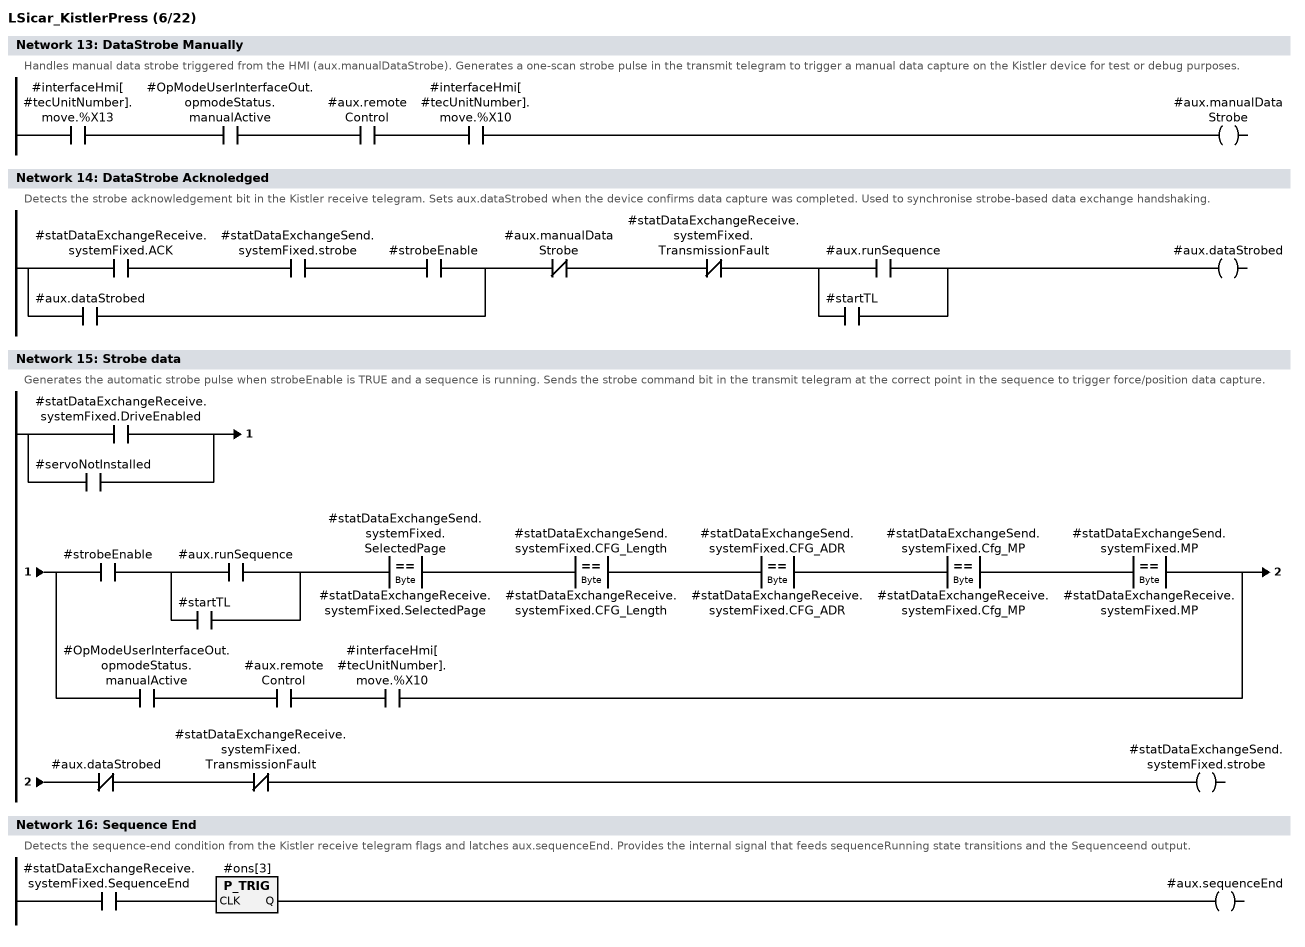
   RUNG wire#powerrail
      Contact( #interfaceHmi[#tecUnitNumber].move.%X13 )
      Contact( #OpModeUserInterfaceOut.opmodeStatus.manualActive )
      Contact( #aux.remoteControl )
      Contact( #interfaceHmi[#tecUnitNumber].move.%X10 )
      Coil( #aux.manualDataStrobe )
   END_RUNG
   // the same network as SCL:
   #aux.manualDataStrobe := #interfaceHmi[#tecUnitNumber].move.%X13 AND #OpModeUserInterfaceOut.opmodeStatus.manualActive AND #aux.remoteControl AND #interfaceHmi[#tecUnitNumber].move.%X10;
END_REGION

REGION Network 14: DataStrobe Acknoledged
   // Detects the strobe acknowledgement bit in the Kistler receive telegram. Sets aux.dataStrobed when the device confirms data capture was completed. Used to synchronise strobe-based data exchange handshaking.
   RUNG wire#powerrail
      Contact( #statDataExchangeReceive.systemFixed.ACK )
      Contact( #statDataExchangeSend.systemFixed.strobe )
      Contact( #strobeEnable )
      wire#w1
      I_Contact( #aux.manualDataStrobe )
      I_Contact( #statDataExchangeReceive.systemFixed.TransmissionFault )
      wire#w2
      Contact( #aux.runSequence )
      wire#w3
      Coil( #aux.dataStrobed )
   END_RUNG
   RUNG wire#powerrail
      Contact( #aux.dataStrobed )
   END_RUNG wire#w1
   RUNG wire#w2
      Contact( #startTL )
   END_RUNG wire#w3
   // the same network as SCL:
   #aux.dataStrobed := ((#statDataExchangeReceive.systemFixed.ACK AND #statDataExchangeSend.systemFixed.strobe AND #strobeEnable) OR #aux.dataStrobed) AND NOT #aux.manualDataStrobe AND NOT #statDataExchangeReceive.systemFixed.TransmissionFault AND (#aux.runSequence OR #startTL);
END_REGION

REGION Network 15: Strobe data
   // Generates the automatic strobe pulse when strobeEnable is TRUE and a sequence is running. Sends the strobe command bit in the transmit telegram at the correct point in the sequence to trigger force/position data capture.
   RUNG wire#powerrail
      Contact( #statDataExchangeReceive.systemFixed.DriveEnabled )
      wire#w1
      Contact( #strobeEnable )
      wire#w2
      Contact( #aux.runSequence )
      wire#w3
      { S7_Templates := "SrcType := Byte" } EQ_Contact(in1 := #statDataExchangeSend.systemFixed.SelectedPage, in2 := #statDataExchangeReceive.systemFixed.SelectedPage)
      { S7_Templates := "SrcType := Byte" } EQ_Contact(in1 := #statDataExchangeSend.systemFixed.CFG_Length, in2 := #statDataExchangeReceive.systemFixed.CFG_Length)
      { S7_Templates := "SrcType := Byte" } EQ_Contact(in1 := #statDataExchangeSend.systemFixed.CFG_ADR, in2 := #statDataExchangeReceive.systemFixed.CFG_ADR)
      { S7_Templates := "SrcType := Byte" } EQ_Contact(in1 := #statDataExchangeSend.systemFixed.Cfg_MP, in2 := #statDataExchangeReceive.systemFixed.Cfg_MP)
      { S7_Templates := "SrcType := Byte" } EQ_Contact(in1 := #statDataExchangeSend.systemFixed.MP, in2 := #statDataExchangeReceive.systemFixed.MP)
      wire#w4
      I_Contact( #aux.dataStrobed )
      I_Contact( #statDataExchangeReceive.systemFixed.TransmissionFault )
      Coil( #statDataExchangeSend.systemFixed.strobe )
   END_RUNG
   RUNG wire#powerrail
      Contact( #servoNotInstalled )
   END_RUNG wire#w1
   RUNG wire#w2
      Contact( #startTL )
   END_RUNG wire#w3
   RUNG wire#w1
      Contact( #OpModeUserInterfaceOut.opmodeStatus.manualActive )
      Contact( #aux.remoteControl )
      Contact( #interfaceHmi[#tecUnitNumber].move.%X10 )
   END_RUNG wire#w4
   // the same network as SCL:
   #statDataExchangeSend.systemFixed.strobe := (#statDataExchangeReceive.systemFixed.DriveEnabled OR #servoNotInstalled) AND ((#strobeEnable AND (#aux.runSequence OR #startTL) AND (#statDataExchangeSend.systemFixed.SelectedPage = #statDataExchangeReceive.systemFixed.SelectedPage) AND (#statDataExchangeSend.systemFixed.CFG_Length = #statDataExchangeReceive.systemFixed.CFG_Length) AND (#statDataExchangeSend.systemFixed.CFG_ADR = #statDataExchangeReceive.systemFixed.CFG_ADR) AND (#statDataExchangeSend.systemFixed.Cfg_MP = #statDataExchangeReceive.systemFixed.Cfg_MP) AND (#statDataExchangeSend.systemFixed.MP = #statDataExchangeReceive.systemFixed.MP)) OR (#OpModeUserInterfaceOut.opmodeStatus.manualActive AND #aux.remoteControl AND #interfaceHmi[#tecUnitNumber].move.%X10)) AND NOT #aux.dataStrobed AND NOT #statDataExchangeReceive.systemFixed.TransmissionFault;
END_REGION

REGION Network 16: Sequence End
   // Detects the sequence-end condition from the Kistler receive telegram flags and latches aux.sequenceEnd. Provides the internal signal that feeds sequenceRunning state transitions and the Sequenceend output.
   RUNG wire#powerrail
      Contact( #statDataExchangeReceive.systemFixed.SequenceEnd )
      P_Trig( #ons[3] )
      Coil( #aux.sequenceEnd )
   END_RUNG
   // the same network as SCL:
   #_w1 := #statDataExchangeReceive.systemFixed.SequenceEnd AND NOT #ons[3];   // rising edge
   #ons[3] := #statDataExchangeReceive.systemFixed.SequenceEnd;
   #aux.sequenceEnd := #_w1;
END_REGION

REGION Network 17: Run the sequence
   // Core sequence start logic. When aux.runSequence is TRUE, no active faults exist, and the block is in automatic mode, triggers the start command in the transmit telegram to begin the Kistler measurement sequence.
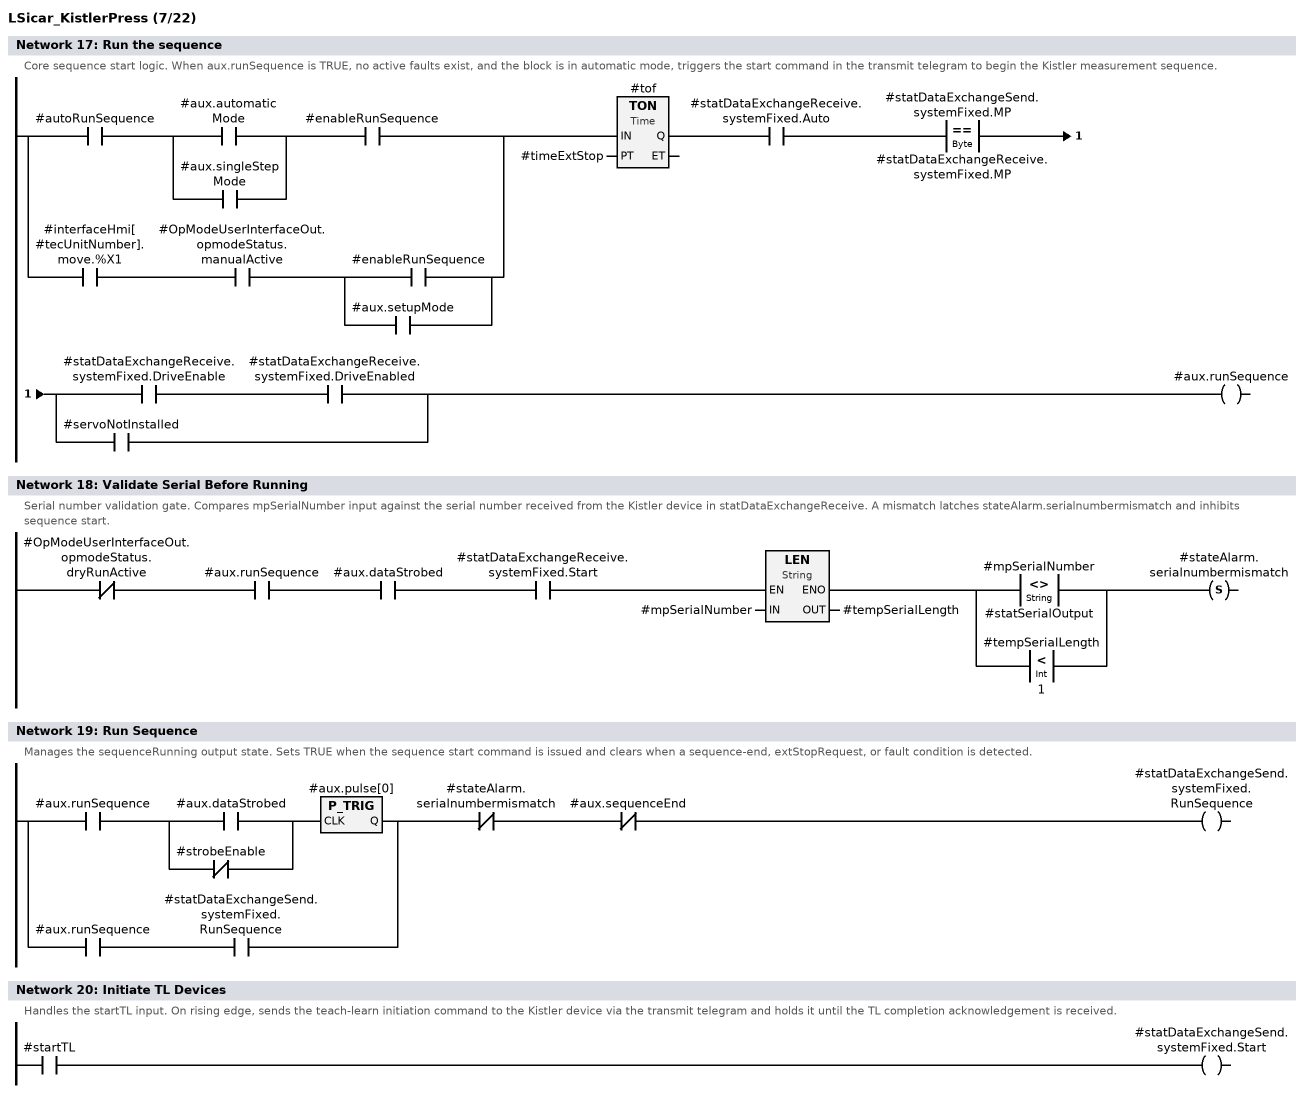
   RUNG wire#powerrail
      Contact( #autoRunSequence )
      wire#w1
      Contact( #aux.automaticMode )
      wire#w2
      Contact( #enableRunSequence )
      wire#w3
      { S7_Templates := "time_type := Time" } #tof.TON(pt := #timeExtStop, et =>)
      Contact( #statDataExchangeReceive.systemFixed.Auto )
      { S7_Templates := "SrcType := Byte" } EQ_Contact(in1 := #statDataExchangeSend.systemFixed.MP, in2 := #statDataExchangeReceive.systemFixed.MP)
      wire#w5
      Contact( #statDataExchangeReceive.systemFixed.DriveEnable )
      Contact( #statDataExchangeReceive.systemFixed.DriveEnabled )
      wire#w6
      Coil( #aux.runSequence )
   END_RUNG
   RUNG wire#w1
      Contact( #aux.singleStepMode )
   END_RUNG wire#w2
   RUNG wire#powerrail
      Contact( #interfaceHmi[#tecUnitNumber].move.%X1 )
      Contact( #OpModeUserInterfaceOut.opmodeStatus.manualActive )
      wire#w4
      Contact( #enableRunSequence )
   END_RUNG wire#w3
   RUNG wire#w4
      Contact( #aux.setupMode )
   END_RUNG wire#w3
   RUNG wire#w5
      Contact( #servoNotInstalled )
   END_RUNG wire#w6
   // the same network as SCL:
   #tof(IN := (#autoRunSequence AND (#aux.automaticMode OR #aux.singleStepMode) AND #enableRunSequence) OR (#interfaceHmi[#tecUnitNumber].move.%X1 AND #OpModeUserInterfaceOut.opmodeStatus.manualActive AND (#enableRunSequence OR #aux.setupMode)),   // TON
        PT := #timeExtStop);
   #aux.runSequence := #tof.Q AND #statDataExchangeReceive.systemFixed.Auto AND (#statDataExchangeSend.systemFixed.MP = #statDataExchangeReceive.systemFixed.MP) AND ((#statDataExchangeReceive.systemFixed.DriveEnable AND #statDataExchangeReceive.systemFixed.DriveEnabled) OR #servoNotInstalled);
END_REGION

REGION Network 18: Validate Serial Before Running
   // Serial number validation gate. Compares mpSerialNumber input against the serial number received from the Kistler device in statDataExchangeReceive. A mismatch latches stateAlarm.serialnumbermismatch and inhibits sequence start.
   RUNG wire#powerrail
      I_Contact( #OpModeUserInterfaceOut.opmodeStatus.dryRunActive )
      Contact( #aux.runSequence )
      Contact( #aux.dataStrobed )
      Contact( #statDataExchangeReceive.systemFixed.Start )
      { S7_Templates := "[str_type := String, return_type := Int]" } LEN(IN := #mpSerialNumber, OUT => #tempSerialLength)
      wire#w1
      { S7_Templates := "SrcType := String" } NE_Contact(in1 := #mpSerialNumber, in2 := #statSerialOutput)
      wire#w2
      S_Coil( #stateAlarm.serialnumbermismatch )
   END_RUNG
   RUNG wire#w1
      { S7_Templates := "SrcType := Int" } LT_Contact(in1 := #tempSerialLength, in2 := 1)
   END_RUNG wire#w2
   // the same network as SCL:
   #_w1 := NOT #OpModeUserInterfaceOut.opmodeStatus.dryRunActive AND #aux.runSequence AND #aux.dataStrobed AND #statDataExchangeReceive.systemFixed.Start;
   LEN(EN := #_w1, IN := #mpSerialNumber, OUT => #tempSerialLength, ENO => #_w2);
   IF #_w2 AND ((#mpSerialNumber <> #statSerialOutput) OR (#tempSerialLength < 1)) THEN
       #stateAlarm.serialnumbermismatch := TRUE;
   END_IF;
END_REGION

REGION Network 19: Run Sequence
   // Manages the sequenceRunning output state. Sets TRUE when the sequence start command is issued and clears when a sequence-end, extStopRequest, or fault condition is detected.
   RUNG wire#powerrail
      Contact( #aux.runSequence )
      wire#w1
      Contact( #aux.dataStrobed )
      wire#w2
      P_Trig( #aux.pulse[0] )
      wire#w3
      I_Contact( #stateAlarm.serialnumbermismatch )
      I_Contact( #aux.sequenceEnd )
      Coil( #statDataExchangeSend.systemFixed.RunSequence )
   END_RUNG
   RUNG wire#w1
      I_Contact( #strobeEnable )
   END_RUNG wire#w2
   RUNG wire#powerrail
      Contact( #aux.runSequence )
      Contact( #statDataExchangeSend.systemFixed.RunSequence )
   END_RUNG wire#w3
   // the same network as SCL:
   #_w1 := #aux.runSequence AND (#aux.dataStrobed OR NOT #strobeEnable);
   #_w2 := #_w1 AND NOT #aux.pulse[0];   // rising edge
   #aux.pulse[0] := #_w1;
   #statDataExchangeSend.systemFixed.RunSequence := (#_w2 OR (#aux.runSequence AND #statDataExchangeSend.systemFixed.RunSequence)) AND NOT #stateAlarm.serialnumbermismatch AND NOT #aux.sequenceEnd;
END_REGION

REGION Network 20: Initiate TL Devices
   // Handles the startTL input. On rising edge, sends the teach-learn initiation command to the Kistler device via the transmit telegram and holds it until the TL completion acknowledgement is received.
   RUNG wire#powerrail
      Contact( #startTL )
      Coil( #statDataExchangeSend.systemFixed.Start )
   END_RUNG
   // the same network as SCL:
   #statDataExchangeSend.systemFixed.Start := #startTL;
END_REGION

REGION Network 21: Monitor Operation Timeouts
   // Runs the operation cycle timer (statInstruction.timeroperation) and other monitoring timers. If timeOperation expires during a running sequence, sets stateAlarm.timerMonitorRunSequence and aborts the cycle.
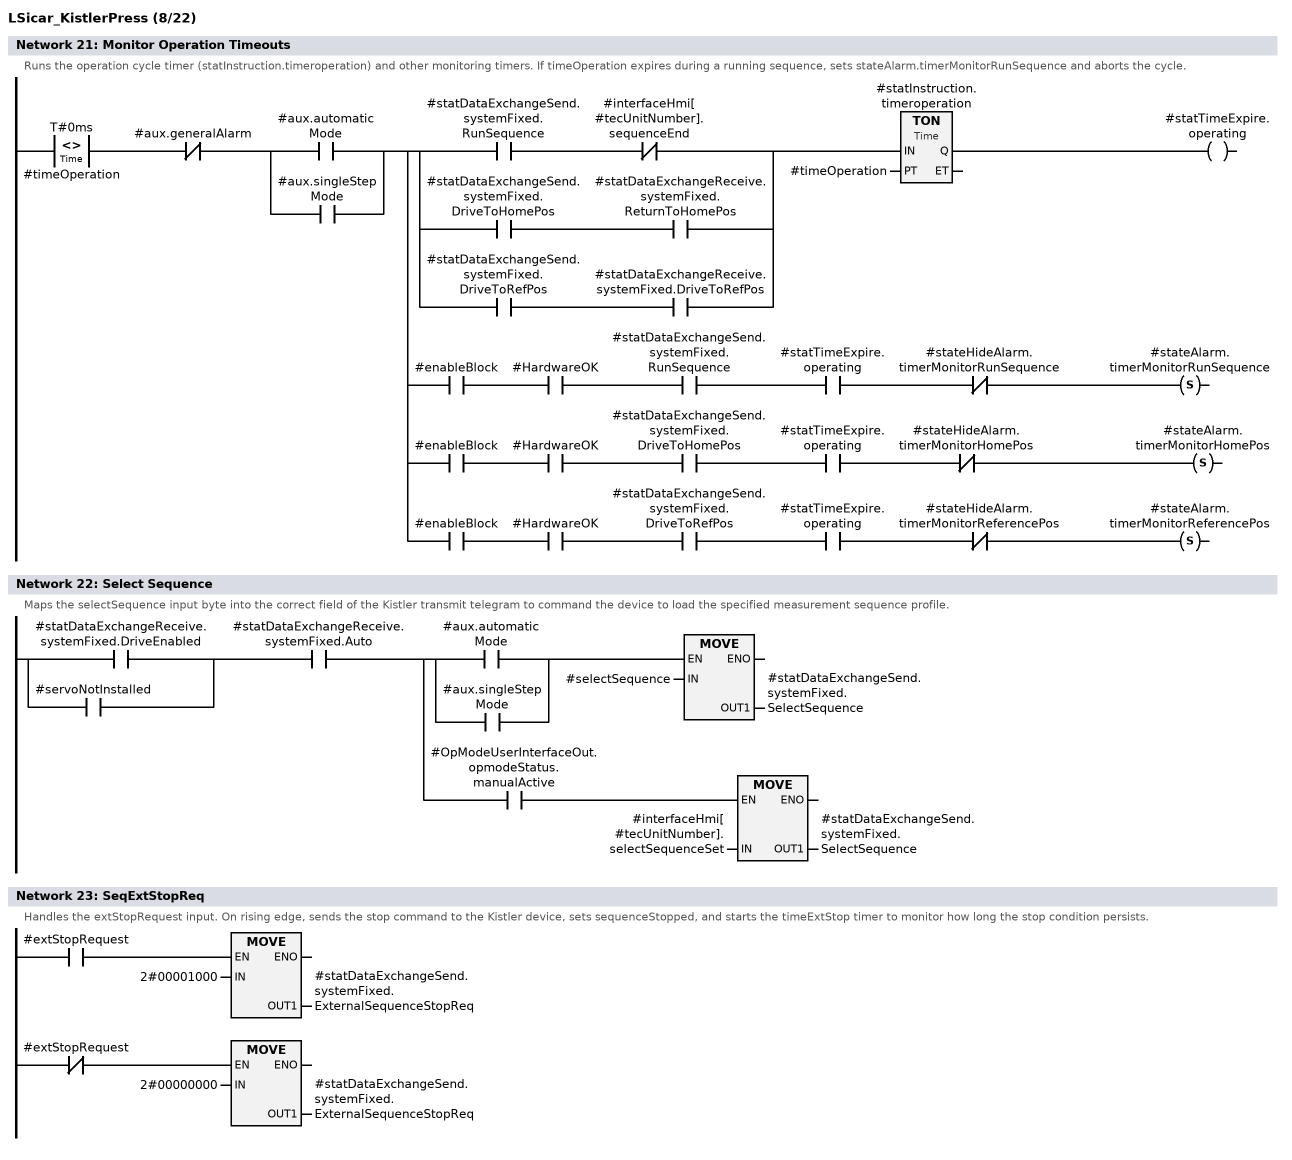
   RUNG wire#powerrail
      { S7_Templates := "SrcType := Time" } NE_Contact(in1 := T#0ms, in2 := #timeOperation)
      I_Contact( #aux.generalAlarm )
      wire#w1
      Contact( #aux.automaticMode )
      wire#w2
      Contact( #statDataExchangeSend.systemFixed.RunSequence )
      I_Contact( #interfaceHmi[#tecUnitNumber].sequenceEnd )
      wire#w3
      { S7_Templates := "time_type := Time" } #statInstruction.timeroperation.TON(pt := #timeOperation, et =>)
      Coil( #statTimeExpire.operating )
   END_RUNG
   RUNG wire#w1
      Contact( #aux.singleStepMode )
   END_RUNG wire#w2
   RUNG wire#w2
      Contact( #statDataExchangeSend.systemFixed.DriveToHomePos )
      Contact( #statDataExchangeReceive.systemFixed.ReturnToHomePos )
   END_RUNG wire#w3
   RUNG wire#w2
      Contact( #statDataExchangeSend.systemFixed.DriveToRefPos )
      Contact( #statDataExchangeReceive.systemFixed.DriveToRefPos )
   END_RUNG wire#w3
   RUNG wire#w2
      Contact( #enableBlock )
      Contact( #HardwareOK )
      Contact( #statDataExchangeSend.systemFixed.RunSequence )
      Contact( #statTimeExpire.operating )
      I_Contact( #stateHideAlarm.timerMonitorRunSequence )
      S_Coil( #stateAlarm.timerMonitorRunSequence )
   END_RUNG
   RUNG wire#w2
      Contact( #enableBlock )
      Contact( #HardwareOK )
      Contact( #statDataExchangeSend.systemFixed.DriveToHomePos )
      Contact( #statTimeExpire.operating )
      I_Contact( #stateHideAlarm.timerMonitorHomePos )
      S_Coil( #stateAlarm.timerMonitorHomePos )
   END_RUNG
   RUNG wire#w2
      Contact( #enableBlock )
      Contact( #HardwareOK )
      Contact( #statDataExchangeSend.systemFixed.DriveToRefPos )
      Contact( #statTimeExpire.operating )
      I_Contact( #stateHideAlarm.timerMonitorReferencePos )
      S_Coil( #stateAlarm.timerMonitorReferencePos )
   END_RUNG
   // the same network as SCL:
   #_w1 := (T#0ms <> #timeOperation) AND NOT #aux.generalAlarm AND (#aux.automaticMode OR #aux.singleStepMode);
   #statInstruction.timeroperation.TON(IN := #_w1 AND ((#statDataExchangeSend.systemFixed.RunSequence AND NOT #interfaceHmi[#tecUnitNumber].sequenceEnd) OR (#statDataExchangeSend.systemFixed.DriveToHomePos AND #statDataExchangeReceive.systemFixed.ReturnToHomePos) OR (#statDataExchangeSend.systemFixed.DriveToRefPos AND #statDataExchangeReceive.systemFixed.DriveToRefPos)),
                           PT := #timeOperation);
   #statTimeExpire.operating := #statInstruction.timeroperation.Q;
   IF #_w1 AND #enableBlock AND #HardwareOK AND #statDataExchangeSend.systemFixed.RunSequence AND #statTimeExpire.operating AND NOT #stateHideAlarm.timerMonitorRunSequence THEN
       #stateAlarm.timerMonitorRunSequence := TRUE;
   END_IF;
   IF #_w1 AND #enableBlock AND #HardwareOK AND #statDataExchangeSend.systemFixed.DriveToHomePos AND #statTimeExpire.operating AND NOT #stateHideAlarm.timerMonitorHomePos THEN
       #stateAlarm.timerMonitorHomePos := TRUE;
   END_IF;
   IF #_w1 AND #enableBlock AND #HardwareOK AND #statDataExchangeSend.systemFixed.DriveToRefPos AND #statTimeExpire.operating AND NOT #stateHideAlarm.timerMonitorReferencePos THEN
       #stateAlarm.timerMonitorReferencePos := TRUE;
   END_IF;
END_REGION

REGION Network 22: Select Sequence
   // Maps the selectSequence input byte into the correct field of the Kistler transmit telegram to command the device to load the specified measurement sequence profile.
   RUNG wire#powerrail
      Contact( #statDataExchangeReceive.systemFixed.DriveEnabled )
      wire#w1
      Contact( #statDataExchangeReceive.systemFixed.Auto )
      wire#w2
      Contact( #aux.automaticMode )
      wire#w3
      Move(in := #selectSequence, out1 => #statDataExchangeSend.systemFixed.SelectSequence)
   END_RUNG
   RUNG wire#powerrail
      Contact( #servoNotInstalled )
   END_RUNG wire#w1
   RUNG wire#w2
      Contact( #aux.singleStepMode )
   END_RUNG wire#w3
   RUNG wire#w2
      Contact( #OpModeUserInterfaceOut.opmodeStatus.manualActive )
      Move(in := #interfaceHmi[#tecUnitNumber].selectSequenceSet, out1 => #statDataExchangeSend.systemFixed.SelectSequence)
   END_RUNG
   // the same network as SCL:
   #_w1 := (#statDataExchangeReceive.systemFixed.DriveEnabled OR #servoNotInstalled) AND #statDataExchangeReceive.systemFixed.Auto;
   IF #_w1 AND (#aux.automaticMode OR #aux.singleStepMode) THEN
       #statDataExchangeSend.systemFixed.SelectSequence := #selectSequence;
   END_IF;
   IF #_w1 AND #OpModeUserInterfaceOut.opmodeStatus.manualActive THEN
       #statDataExchangeSend.systemFixed.SelectSequence := #interfaceHmi[#tecUnitNumber].selectSequenceSet;
   END_IF;
END_REGION

REGION Network 23: SeqExtStopReq
   // Handles the extStopRequest input. On rising edge, sends the stop command to the Kistler device, sets sequenceStopped, and starts the timeExtStop timer to monitor how long the stop condition persists.
   RUNG wire#powerrail
      Contact( #extStopRequest )
      Move(in := 2#00001000, out1 => #statDataExchangeSend.systemFixed.ExternalSequenceStopReq)
   END_RUNG
   RUNG wire#powerrail
      I_Contact( #extStopRequest )
      Move(in := 2#00000000, out1 => #statDataExchangeSend.systemFixed.ExternalSequenceStopReq)
   END_RUNG
   // the same network as SCL:
   IF #extStopRequest THEN #statDataExchangeSend.systemFixed.ExternalSequenceStopReq := 2#00001000; END_IF;
   IF NOT #extStopRequest THEN
       #statDataExchangeSend.systemFixed.ExternalSequenceStopReq := 2#00000000;
   END_IF;
END_REGION

REGION Network 24: Resume After Error
   // Resume after error. On rising edge of continuewait input, clears the waitContinue pause flag and allows the sequence to continue. Sends the continue command to the Kistler device and clears any latched soft-stop faults.
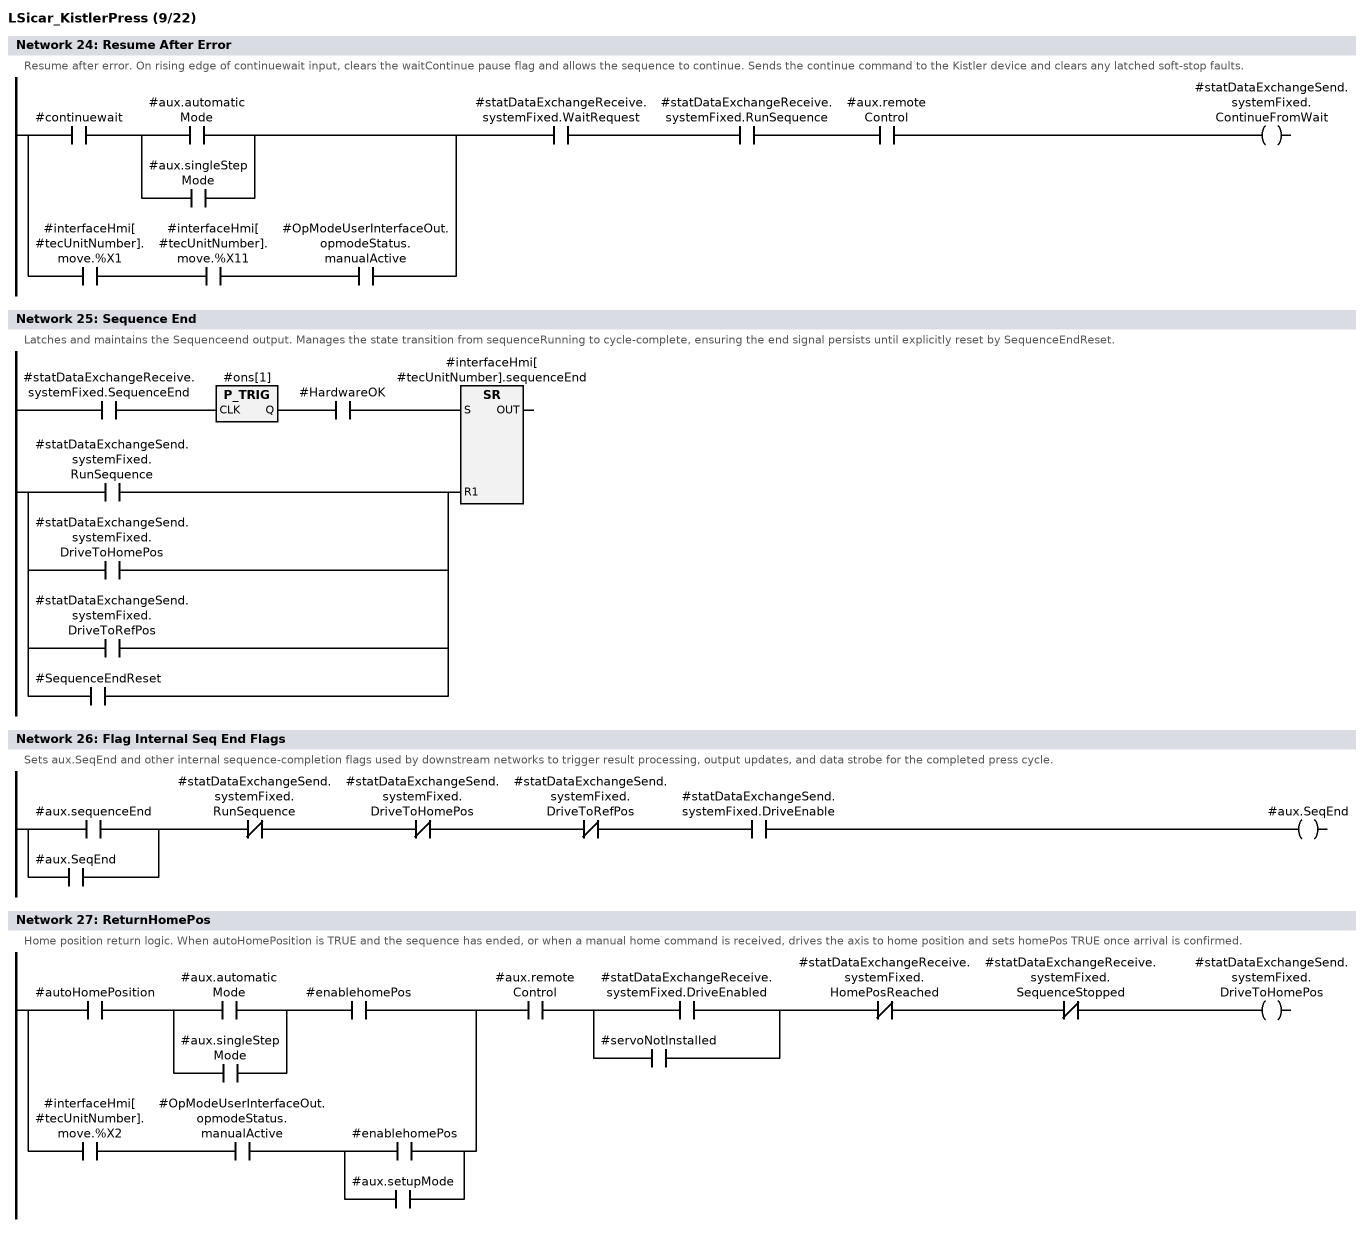
   RUNG wire#powerrail
      Contact( #continuewait )
      wire#w1
      Contact( #aux.automaticMode )
      wire#w2
      Contact( #statDataExchangeReceive.systemFixed.WaitRequest )
      Contact( #statDataExchangeReceive.systemFixed.RunSequence )
      Contact( #aux.remoteControl )
      Coil( #statDataExchangeSend.systemFixed.ContinueFromWait )
   END_RUNG
   RUNG wire#w1
      Contact( #aux.singleStepMode )
   END_RUNG wire#w2
   RUNG wire#powerrail
      Contact( #interfaceHmi[#tecUnitNumber].move.%X1 )
      Contact( #interfaceHmi[#tecUnitNumber].move.%X11 )
      Contact( #OpModeUserInterfaceOut.opmodeStatus.manualActive )
   END_RUNG wire#w2
   // the same network as SCL:
   #statDataExchangeSend.systemFixed.ContinueFromWait := ((#continuewait AND (#aux.automaticMode OR #aux.singleStepMode)) OR (#interfaceHmi[#tecUnitNumber].move.%X1 AND #interfaceHmi[#tecUnitNumber].move.%X11 AND #OpModeUserInterfaceOut.opmodeStatus.manualActive)) AND #statDataExchangeReceive.systemFixed.WaitRequest AND #statDataExchangeReceive.systemFixed.RunSequence AND #aux.remoteControl;
END_REGION

REGION Network 25: Sequence End
   // Latches and maintains the Sequenceend output. Manages the state transition from sequenceRunning to cycle-complete, ensuring the end signal persists until explicitly reset by SequenceEndReset.
   RUNG wire#powerrail
      Contact( #statDataExchangeReceive.systemFixed.SequenceEnd )
      P_Trig( #ons[1] )
      Contact( #HardwareOK )
      S_SR(operand := #interfaceHmi[#tecUnitNumber].sequenceEnd, r1 := wire#w1)
   END_RUNG
   RUNG wire#powerrail
      Contact( #statDataExchangeSend.systemFixed.RunSequence )
   END_RUNG wire#w1
   RUNG wire#powerrail
      Contact( #statDataExchangeSend.systemFixed.DriveToHomePos )
   END_RUNG wire#w1
   RUNG wire#powerrail
      Contact( #statDataExchangeSend.systemFixed.DriveToRefPos )
   END_RUNG wire#w1
   RUNG wire#powerrail
      Contact( #SequenceEndReset )
   END_RUNG wire#w1
   // the same network as SCL:
   #_w1 := #statDataExchangeReceive.systemFixed.SequenceEnd AND NOT #ons[1];   // rising edge
   #ons[1] := #statDataExchangeReceive.systemFixed.SequenceEnd;
   IF #_w1 AND #HardwareOK THEN
       #interfaceHmi[#tecUnitNumber].sequenceEnd := TRUE;   // SR flip-flop
   END_IF;
   IF #statDataExchangeSend.systemFixed.RunSequence OR #statDataExchangeSend.systemFixed.DriveToHomePos OR #statDataExchangeSend.systemFixed.DriveToRefPos OR #SequenceEndReset THEN
       #interfaceHmi[#tecUnitNumber].sequenceEnd := FALSE;
   END_IF;
END_REGION

REGION Network 26: Flag Internal Seq End Flags
   // Sets aux.SeqEnd and other internal sequence-completion flags used by downstream networks to trigger result processing, output updates, and data strobe for the completed press cycle.
   RUNG wire#powerrail
      Contact( #aux.sequenceEnd )
      wire#w1
      I_Contact( #statDataExchangeSend.systemFixed.RunSequence )
      I_Contact( #statDataExchangeSend.systemFixed.DriveToHomePos )
      I_Contact( #statDataExchangeSend.systemFixed.DriveToRefPos )
      Contact( #statDataExchangeSend.systemFixed.DriveEnable )
      Coil( #aux.SeqEnd )
   END_RUNG
   RUNG wire#powerrail
      Contact( #aux.SeqEnd )
   END_RUNG wire#w1
   // the same network as SCL:
   #aux.SeqEnd := (#aux.sequenceEnd OR #aux.SeqEnd) AND NOT #statDataExchangeSend.systemFixed.RunSequence AND NOT #statDataExchangeSend.systemFixed.DriveToHomePos AND NOT #statDataExchangeSend.systemFixed.DriveToRefPos AND #statDataExchangeSend.systemFixed.DriveEnable;
END_REGION

REGION Network 27: ReturnHomePos
   // Home position return logic. When autoHomePosition is TRUE and the sequence has ended, or when a manual home command is received, drives the axis to home position and sets homePos TRUE once arrival is confirmed.
   RUNG wire#powerrail
      Contact( #autoHomePosition )
      wire#w1
      Contact( #aux.automaticMode )
      wire#w2
      Contact( #enablehomePos )
      wire#w3
      Contact( #aux.remoteControl )
      wire#w5
      Contact( #statDataExchangeReceive.systemFixed.DriveEnabled )
      wire#w6
      I_Contact( #statDataExchangeReceive.systemFixed.HomePosReached )
      I_Contact( #statDataExchangeReceive.systemFixed.SequenceStopped )
      Coil( #statDataExchangeSend.systemFixed.DriveToHomePos )
   END_RUNG
   RUNG wire#w1
      Contact( #aux.singleStepMode )
   END_RUNG wire#w2
   RUNG wire#powerrail
      Contact( #interfaceHmi[#tecUnitNumber].move.%X2 )
      Contact( #OpModeUserInterfaceOut.opmodeStatus.manualActive )
      wire#w4
      Contact( #enablehomePos )
   END_RUNG wire#w3
   RUNG wire#w4
      Contact( #aux.setupMode )
   END_RUNG wire#w3
   RUNG wire#w5
      Contact( #servoNotInstalled )
   END_RUNG wire#w6
   // the same network as SCL:
   #statDataExchangeSend.systemFixed.DriveToHomePos := ((#autoHomePosition AND (#aux.automaticMode OR #aux.singleStepMode) AND #enablehomePos) OR (#interfaceHmi[#tecUnitNumber].move.%X2 AND #OpModeUserInterfaceOut.opmodeStatus.manualActive AND (#enablehomePos OR #aux.setupMode))) AND #aux.remoteControl AND (#statDataExchangeReceive.systemFixed.DriveEnabled OR #servoNotInstalled) AND NOT #statDataExchangeReceive.systemFixed.HomePosReached AND NOT #statDataExchangeReceive.systemFixed.SequenceStopped;
END_REGION

REGION Network 28: DrivetoRefPOs
   // Reference position drive logic. When autoDriveToReferencePosition is TRUE at startup/reset, or on a manual reference command, drives the axis to the calibration reference position and sets referencePos TRUE on arrival.
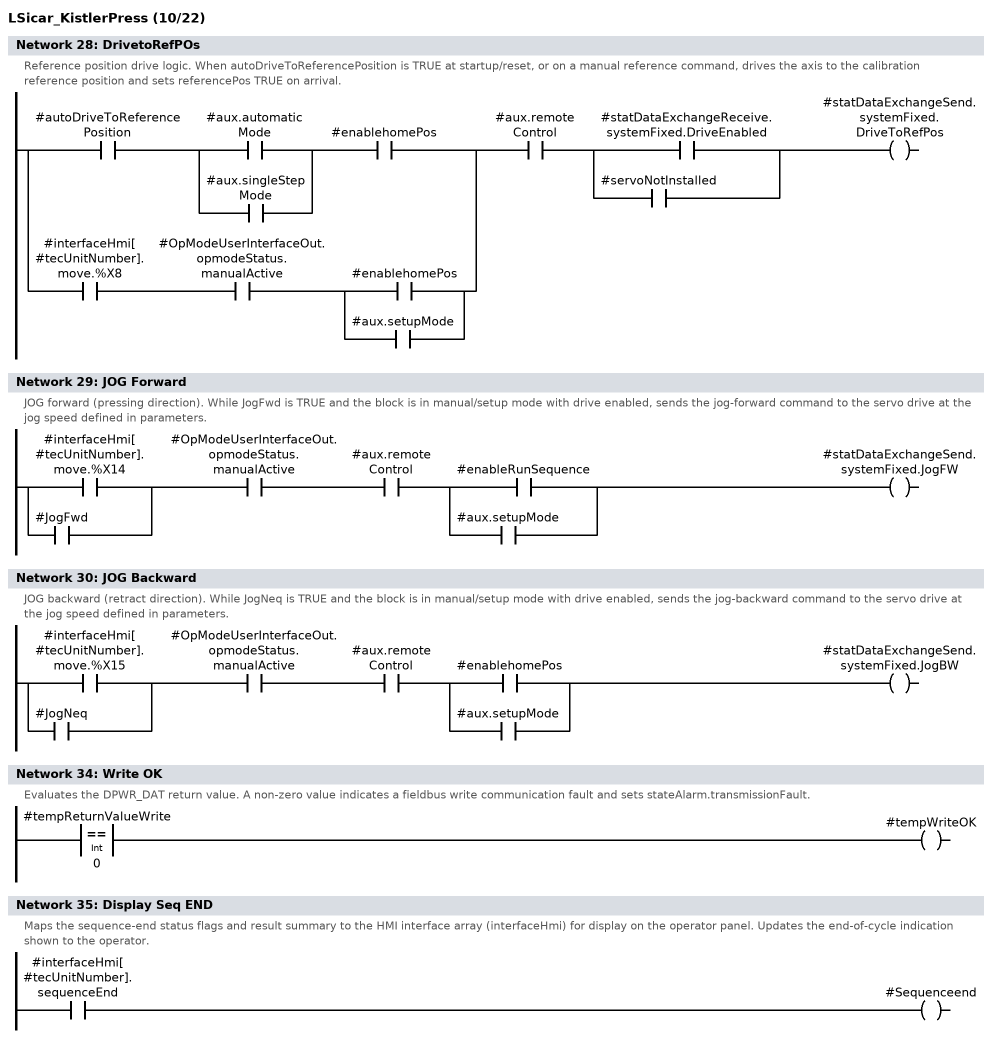
   RUNG wire#powerrail
      Contact( #autoDriveToReferencePosition )
      wire#w1
      Contact( #aux.automaticMode )
      wire#w2
      Contact( #enablehomePos )
      wire#w3
      Contact( #aux.remoteControl )
      wire#w5
      Contact( #statDataExchangeReceive.systemFixed.DriveEnabled )
      wire#w6
      Coil( #statDataExchangeSend.systemFixed.DriveToRefPos )
   END_RUNG
   RUNG wire#w1
      Contact( #aux.singleStepMode )
   END_RUNG wire#w2
   RUNG wire#powerrail
      Contact( #interfaceHmi[#tecUnitNumber].move.%X8 )
      Contact( #OpModeUserInterfaceOut.opmodeStatus.manualActive )
      wire#w4
      Contact( #enablehomePos )
   END_RUNG wire#w3
   RUNG wire#w4
      Contact( #aux.setupMode )
   END_RUNG wire#w3
   RUNG wire#w5
      Contact( #servoNotInstalled )
   END_RUNG wire#w6
   // the same network as SCL:
   #statDataExchangeSend.systemFixed.DriveToRefPos := ((#autoDriveToReferencePosition AND (#aux.automaticMode OR #aux.singleStepMode) AND #enablehomePos) OR (#interfaceHmi[#tecUnitNumber].move.%X8 AND #OpModeUserInterfaceOut.opmodeStatus.manualActive AND (#enablehomePos OR #aux.setupMode))) AND #aux.remoteControl AND (#statDataExchangeReceive.systemFixed.DriveEnabled OR #servoNotInstalled);
END_REGION

REGION Network 29: JOG Forward
   // JOG forward (pressing direction). While JogFwd is TRUE and the block is in manual/setup mode with drive enabled, sends the jog-forward command to the servo drive at the jog speed defined in parameters.
   RUNG wire#powerrail
      Contact( #interfaceHmi[#tecUnitNumber].move.%X14 )
      wire#w1
      Contact( #OpModeUserInterfaceOut.opmodeStatus.manualActive )
      Contact( #aux.remoteControl )
      wire#w2
      Contact( #enableRunSequence )
      wire#w3
      Coil( #statDataExchangeSend.systemFixed.JogFW )
   END_RUNG
   RUNG wire#powerrail
      Contact( #JogFwd )
   END_RUNG wire#w1
   RUNG wire#w2
      Contact( #aux.setupMode )
   END_RUNG wire#w3
   // the same network as SCL:
   #statDataExchangeSend.systemFixed.JogFW := (#interfaceHmi[#tecUnitNumber].move.%X14 OR #JogFwd) AND #OpModeUserInterfaceOut.opmodeStatus.manualActive AND #aux.remoteControl AND (#enableRunSequence OR #aux.setupMode);
END_REGION

REGION Network 30: JOG Backward
   // JOG backward (retract direction). While JogNeq is TRUE and the block is in manual/setup mode with drive enabled, sends the jog-backward command to the servo drive at the jog speed defined in parameters.
   RUNG wire#powerrail
      Contact( #interfaceHmi[#tecUnitNumber].move.%X15 )
      wire#w1
      Contact( #OpModeUserInterfaceOut.opmodeStatus.manualActive )
      Contact( #aux.remoteControl )
      wire#w2
      Contact( #enablehomePos )
      wire#w3
      Coil( #statDataExchangeSend.systemFixed.JogBW )
   END_RUNG
   RUNG wire#powerrail
      Contact( #JogNeq )
   END_RUNG wire#w1
   RUNG wire#w2
      Contact( #aux.setupMode )
   END_RUNG wire#w3
   // the same network as SCL:
   #statDataExchangeSend.systemFixed.JogBW := (#interfaceHmi[#tecUnitNumber].move.%X15 OR #JogNeq) AND #OpModeUserInterfaceOut.opmodeStatus.manualActive AND #aux.remoteControl AND (#enablehomePos OR #aux.setupMode);
END_REGION

REGION Network 31 (SCL): Map Incoming Field Bus data for the 200 bytes
   // Extracts individual status flags, result bytes, and diagnostic words from the 200-byte statDataExchangeReceive buffer into named members of the aux and stateAlarm structs for use by control and alarm networks.
   // Jog Speed
   #tempValue := SWAP(REAL_TO_DWORD(#interfaceHmi[#tecUnitNumber].serverJogSpeedSet));
   #statDataExchangeSend.userDefinedOutData[20] := #tempValue.%B0;
   #statDataExchangeSend.userDefinedOutData[21] := #tempValue.%B1;
   #statDataExchangeSend.userDefinedOutData[22] := #tempValue.%B2;
   #statDataExchangeSend.userDefinedOutData[23] := #tempValue.%B3;

   // Jog Max Force
   #tempValue := SWAP(REAL_TO_DWORD(#interfaceHmi[#tecUnitNumber].serverJogMaxForceSet));
   #statDataExchangeSend.userDefinedOutData[24] := #tempValue.%B0;
   #statDataExchangeSend.userDefinedOutData[25] := #tempValue.%B1;
   #statDataExchangeSend.userDefinedOutData[26] := #tempValue.%B2;
   #statDataExchangeSend.userDefinedOutData[27] := #tempValue.%B3;

   // Serial Number
   #tempString := #mpSerialNumber;
   FOR #statSerialByteIndex := 28 TO 51 DO
       #statStringIndex := #statSerialByteIndex - 27;
       #statDataExchangeSend.userDefinedOutData[#statSerialByteIndex] := CHAR_TO_BYTE(#tempString[#statStringIndex]);
   END_FOR;

   // Universal Variables
   #tempDint := 32;
   FOR #i := 0 TO 9 DO
       #tempDword := REAL_TO_DWORD(#parameters.universalvariables[#i]);
       #tempErrorValue := Serialize(SRC_VARIABLE := #tempDword,
                                    DEST_ARRAY => #statDataExchangeSend.userDefinedOutData,
                                    POS := #tempDint);
       #tempDint := #tempDint + 4;
   END_FOR;
END_REGION

REGION Network 32 (SCL): Map Digital Signals
   // Maps boolean signal bits from the Kistler fieldbus receive telegram bitfield words into named boolean members of the statDataExchangeReceive structure for clean access by downstream logic networks.
   #statDataExchangeSend.systemFixed.UNI0 := #parameters.UNI_in[0];
   #statDataExchangeSend.systemFixed.UNI1 := #parameters.UNI_in[1];
   #statDataExchangeSend.systemFixed.UNI2 := #parameters.UNI_in[2];
   #statDataExchangeSend.systemFixed.UNI3 := #parameters.UNI_in[3];
   #statDataExchangeSend.systemFixed.UNI4 := #parameters.UNI_in[4];
   #statDataExchangeSend.systemFixed.UNI5 := #parameters.UNI_in[5];
   #statDataExchangeSend.systemFixed.UNI6 := #parameters.UNI_in[6];
   #statDataExchangeSend.systemFixed.UNI7 := #parameters.UNI_in[7];
END_REGION

REGION Network 33 (SCL): Write Raw Data to Kislter
   // DPWR_DAT writes the statDataExchangeSend transmit telegram to the secondary Kistler PROFINET device (hardwareID2). Called every scan to continuously update the device with current commands and configuration.
       #tempReturnValueWrite := DPWR_DAT(LADDR := #hardwareID2, RECORD:= #statDataExchangeSend);    // Read from Kistler
END_REGION

REGION Network 34: Write OK
   // Evaluates the DPWR_DAT return value. A non-zero value indicates a fieldbus write communication fault and sets stateAlarm.transmissionFault.
   RUNG wire#powerrail
      { S7_Templates := "SrcType := Int" } EQ_Contact(in1 := #tempReturnValueWrite, in2 := 0)
      Coil( #tempWriteOK )
   END_RUNG
   // the same network as SCL:
   #tempWriteOK := #tempReturnValueWrite = 0;
END_REGION

REGION Network 35: Display Seq END
   // Maps the sequence-end status flags and result summary to the HMI interface array (interfaceHmi) for display on the operator panel. Updates the end-of-cycle indication shown to the operator.
   RUNG wire#powerrail
      Contact( #interfaceHmi[#tecUnitNumber].sequenceEnd )
      Coil( #Sequenceend )
   END_RUNG
   // the same network as SCL:
   #Sequenceend := #interfaceHmi[#tecUnitNumber].sequenceEnd;
END_REGION

REGION Network 36: Map Fixed Fieldbus outputs to internal flags
   // Writes the fixed/static fieldbus output bytes that must always be present in the transmit telegram regardless of sequence state. These include protocol control bytes, enable flags, and constant configuration words.
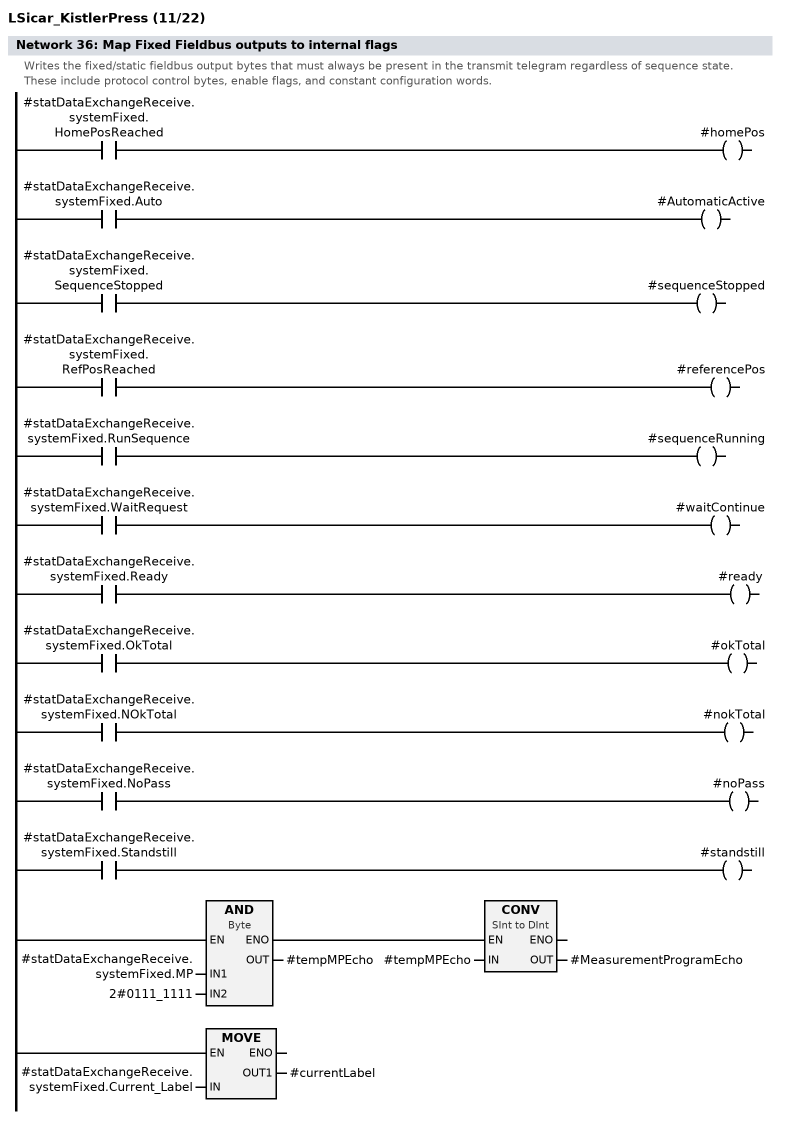
   RUNG wire#powerrail
      Contact( #statDataExchangeReceive.systemFixed.HomePosReached )
      Coil( #homePos )
   END_RUNG
   RUNG wire#powerrail
      Contact( #statDataExchangeReceive.systemFixed.Auto )
      Coil( #AutomaticActive )
   END_RUNG
   RUNG wire#powerrail
      Contact( #statDataExchangeReceive.systemFixed.SequenceStopped )
      Coil( #sequenceStopped )
   END_RUNG
   RUNG wire#powerrail
      Contact( #statDataExchangeReceive.systemFixed.RefPosReached )
      Coil( #referencePos )
   END_RUNG
   RUNG wire#powerrail
      Contact( #statDataExchangeReceive.systemFixed.RunSequence )
      Coil( #sequenceRunning )
   END_RUNG
   RUNG wire#powerrail
      Contact( #statDataExchangeReceive.systemFixed.WaitRequest )
      Coil( #waitContinue )
   END_RUNG
   RUNG wire#powerrail
      Contact( #statDataExchangeReceive.systemFixed.Ready )
      Coil( #ready )
   END_RUNG
   RUNG wire#powerrail
      Contact( #statDataExchangeReceive.systemFixed.OkTotal )
      Coil( #okTotal )
   END_RUNG
   RUNG wire#powerrail
      Contact( #statDataExchangeReceive.systemFixed.NOkTotal )
      Coil( #nokTotal )
   END_RUNG
   RUNG wire#powerrail
      Contact( #statDataExchangeReceive.systemFixed.NoPass )
      Coil( #noPass )
   END_RUNG
   RUNG wire#powerrail
      Contact( #statDataExchangeReceive.systemFixed.Standstill )
      Coil( #standstill )
   END_RUNG
   RUNG wire#powerrail
      { S7_Templates := "SrcType := Byte" } And(in1 := #statDataExchangeReceive.systemFixed.MP, in2 := 2#0111_1111, out => #tempMPEcho)
      { S7_Templates := "[SrcType := SInt, DestType := DInt]" } Convert(in := #tempMPEcho, out => #MeasurementProgramEcho)
   END_RUNG
   RUNG wire#powerrail
      Move(in := #statDataExchangeReceive.systemFixed.Current_Label, out1 => #currentLabel)
   END_RUNG
   // the same network as SCL:
   #homePos := #statDataExchangeReceive.systemFixed.HomePosReached;
   #AutomaticActive := #statDataExchangeReceive.systemFixed.Auto;
   #sequenceStopped := #statDataExchangeReceive.systemFixed.SequenceStopped;
   #referencePos := #statDataExchangeReceive.systemFixed.RefPosReached;
   #sequenceRunning := #statDataExchangeReceive.systemFixed.RunSequence;
   #waitContinue := #statDataExchangeReceive.systemFixed.WaitRequest;
   #ready := #statDataExchangeReceive.systemFixed.Ready;
   #okTotal := #statDataExchangeReceive.systemFixed.OkTotal;
   #nokTotal := #statDataExchangeReceive.systemFixed.NOkTotal;
   #noPass := #statDataExchangeReceive.systemFixed.NoPass;
   #standstill := #statDataExchangeReceive.systemFixed.Standstill;
   #tempMPEcho := #statDataExchangeReceive.systemFixed.MP AND 2#0111_1111;
   #MeasurementProgramEcho := SINT_TO_DINT(#tempMPEcho);
   #currentLabel := #statDataExchangeReceive.systemFixed.Current_Label;
END_REGION

REGION Network 37 (SCL): Process Values Mapping
   // Scales raw fieldbus receive data into engineering units and maps to pvCurrentValueX (position mm), pvCurrentValueY (force kN), pvCurveXminX/XmaxX, pvCurveYminY/YmaxY, and the full customeProcessValues struct.
   // Current Value X
   #tempValue.%B0 := #statDataExchangeReceive.userDefinedOutData[20];
   #tempValue.%B1 := #statDataExchangeReceive.userDefinedOutData[21];
   #tempValue.%B2 := #statDataExchangeReceive.userDefinedOutData[22];
   #tempValue.%B3 := #statDataExchangeReceive.userDefinedOutData[23];
   #pvCurrentValueX := DWORD_TO_REAL(SWAP(#tempValue));

   // Current Value Y
   #tempValue.%B0 := #statDataExchangeReceive.userDefinedOutData[24];
   #tempValue.%B1 := #statDataExchangeReceive.userDefinedOutData[25];
   #tempValue.%B2 := #statDataExchangeReceive.userDefinedOutData[26];
   #tempValue.%B3 := #statDataExchangeReceive.userDefinedOutData[27];
   #pvCurrentValueY := DWORD_TO_REAL(SWAP(#tempValue));

   // Serial Number
   FOR #statSerialByteIndex := 40 TO 63 DO
       #statStringIndex := #statSerialByteIndex - 39;
       #tempString[#statStringIndex] := BYTE_TO_CHAR(#statDataExchangeReceive.userDefinedOutData[#statSerialByteIndex]);
   END_FOR;
   #statSerialOutput := #tempString;

   // Curve XminX
   #tempValue.%B0 := #statDataExchangeReceive.userDefinedOutData[64];
   #tempValue.%B1 := #statDataExchangeReceive.userDefinedOutData[65];
   #tempValue.%B2 := #statDataExchangeReceive.userDefinedOutData[66];
   #tempValue.%B3 := #statDataExchangeReceive.userDefinedOutData[67];
   #pvCurveXminX := DWORD_TO_REAL(SWAP(#tempValue));

   // Curve XmaxX
   #tempValue.%B0 := #statDataExchangeReceive.userDefinedOutData[68];
   #tempValue.%B1 := #statDataExchangeReceive.userDefinedOutData[69];
   #tempValue.%B2 := #statDataExchangeReceive.userDefinedOutData[70];
   #tempValue.%B3 := #statDataExchangeReceive.userDefinedOutData[71];
   #pvCurveXmaxX := DWORD_TO_REAL(SWAP(#tempValue));

   // Curve YminY
   #tempValue.%B0 := #statDataExchangeReceive.userDefinedOutData[72];
   #tempValue.%B1 := #statDataExchangeReceive.userDefinedOutData[73];
   #tempValue.%B2 := #statDataExchangeReceive.userDefinedOutData[74];
   #tempValue.%B3 := #statDataExchangeReceive.userDefinedOutData[75];
   #pvCurveYminY := DWORD_TO_REAL(SWAP(#tempValue));

   // Curve YmaxY
   #tempValue.%B0 := #statDataExchangeReceive.userDefinedOutData[76];
   #tempValue.%B1 := #statDataExchangeReceive.userDefinedOutData[77];
   #tempValue.%B2 := #statDataExchangeReceive.userDefinedOutData[78];
   #tempValue.%B3 := #statDataExchangeReceive.userDefinedOutData[79];
   #pvCurveYmaxY := DWORD_TO_REAL(SWAP(#tempValue));

   // E01 Force
   #tempValue.%B0 := #statDataExchangeReceive.userDefinedOutData[96];
   #tempValue.%B1 := #statDataExchangeReceive.userDefinedOutData[97];
   #tempValue.%B2 := #statDataExchangeReceive.userDefinedOutData[98];
   #tempValue.%B3 := #statDataExchangeReceive.userDefinedOutData[99];
   #customeProcessValues.pv1Force := DWORD_TO_REAL(SWAP(#tempValue));

   // E02 Distance
   #tempValue.%B0 := #statDataExchangeReceive.userDefinedOutData[100];
   #tempValue.%B1 := #statDataExchangeReceive.userDefinedOutData[101];
   #tempValue.%B2 := #statDataExchangeReceive.userDefinedOutData[102];
   #tempValue.%B3 := #statDataExchangeReceive.userDefinedOutData[103];
   #customeProcessValues.pv2Distance := DWORD_TO_REAL(SWAP(#tempValue));

   // E03 Gradient
   #tempValue.%B0 := #statDataExchangeReceive.userDefinedOutData[104];
   #tempValue.%B1 := #statDataExchangeReceive.userDefinedOutData[105];
   #tempValue.%B2 := #statDataExchangeReceive.userDefinedOutData[106];
   #tempValue.%B3 := #statDataExchangeReceive.userDefinedOutData[107];
   #customeProcessValues.pv3Gradient := DWORD_TO_REAL(SWAP(#tempValue));

   // E04 Nopass
   #customeProcessValues.pv4Nopass := #statDataExchangeReceive.userDefinedOutData[108];

   // E05 Unibox
   #customeProcessValues.pv5Unibox := #statDataExchangeReceive.userDefinedOutData[109];

   // E06 Envelope
   #customeProcessValues.pv6Envelope := #statDataExchangeReceive.userDefinedOutData[110];

   // E07 Real
   #tempValue.%B0 := #statDataExchangeReceive.userDefinedOutData[111];
   #tempValue.%B1 := #statDataExchangeReceive.userDefinedOutData[112];
   #tempValue.%B2 := #statDataExchangeReceive.userDefinedOutData[113];
   #tempValue.%B3 := #statDataExchangeReceive.userDefinedOutData[114];
   #customeProcessValues.pv7Real := DWORD_TO_REAL(SWAP(#tempValue));

   // E08 Real
   #tempValue.%B0 := #statDataExchangeReceive.userDefinedOutData[115];
   #tempValue.%B1 := #statDataExchangeReceive.userDefinedOutData[116];
   #tempValue.%B2 := #statDataExchangeReceive.userDefinedOutData[117];
   #tempValue.%B3 := #statDataExchangeReceive.userDefinedOutData[118];
   #customeProcessValues.pv8Real := DWORD_TO_REAL(SWAP(#tempValue));

   // E09 Real
   #tempValue.%B0 := #statDataExchangeReceive.userDefinedOutData[119];
   #tempValue.%B1 := #statDataExchangeReceive.userDefinedOutData[120];
   #tempValue.%B2 := #statDataExchangeReceive.userDefinedOutData[121];
   #tempValue.%B3 := #statDataExchangeReceive.userDefinedOutData[122];
   #customeProcessValues.pv9Real := DWORD_TO_REAL(SWAP(#tempValue));

   // E010 Real
   #tempValue.%B0 := #statDataExchangeReceive.userDefinedOutData[123];
   #tempValue.%B1 := #statDataExchangeReceive.userDefinedOutData[124];
   #tempValue.%B2 := #statDataExchangeReceive.userDefinedOutData[125];
   #tempValue.%B3 := #statDataExchangeReceive.userDefinedOutData[126];
   #customeProcessValues.pv10Real := DWORD_TO_REAL(SWAP(#tempValue));

   // E07 Byte
   #customeProcessValues.pv7Byte := #statDataExchangeReceive.userDefinedOutData[142];

   // E08 Byte
   #customeProcessValues.pv8Byte := #statDataExchangeReceive.userDefinedOutData[143];

   // E09 Byte
   #customeProcessValues.pv9Byte := #statDataExchangeReceive.userDefinedOutData[144];

   // E010 Byte
   #customeProcessValues.pv10Byte := #statDataExchangeReceive.userDefinedOutData[145];
END_REGION

REGION Network 38: Alarms
   // Evaluates all stateAlarm struct bits against the corresponding stateHideAlarm mask bits and the global hideAlarmAll flag. Produces the final set of visible alarm conditions used by Evaluate Internal Alarms and Fault General Alarm.
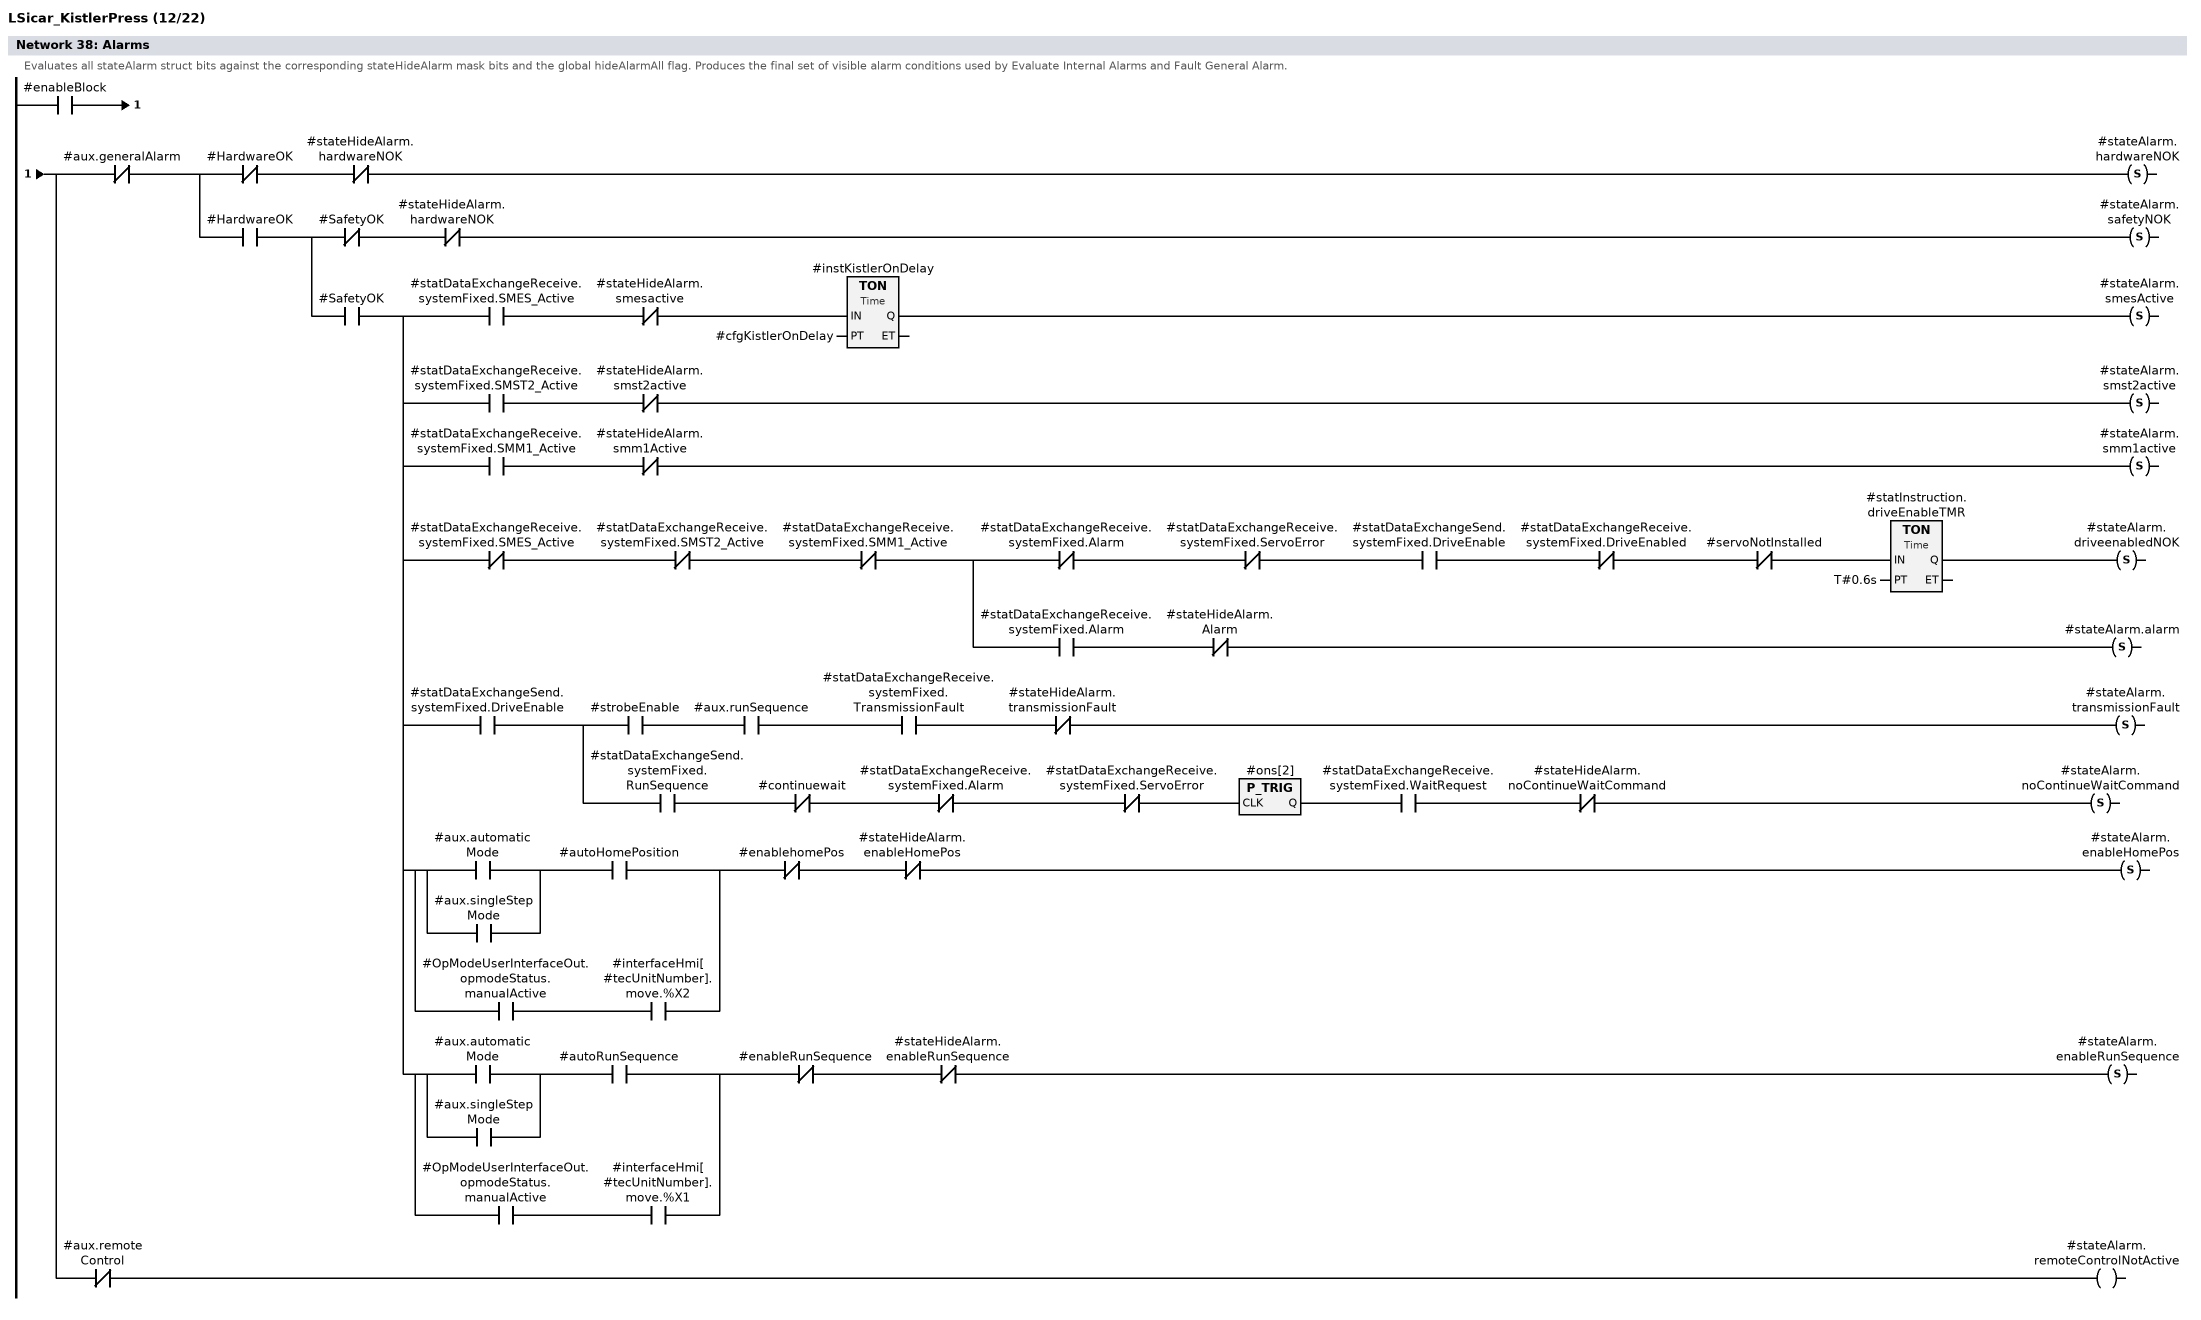
   RUNG wire#powerrail
      Contact( #enableBlock )
      wire#w1
      I_Contact( #aux.generalAlarm )
      wire#w2
      I_Contact( #HardwareOK )
      I_Contact( #stateHideAlarm.hardwareNOK )
      S_Coil( #stateAlarm.hardwareNOK )
   END_RUNG
   RUNG wire#w2
      Contact( #HardwareOK )
      wire#w3
      I_Contact( #SafetyOK )
      I_Contact( #stateHideAlarm.hardwareNOK )
      S_Coil( #stateAlarm.safetyNOK )
   END_RUNG
   RUNG wire#w3
      Contact( #SafetyOK )
      wire#w4
      Contact( #statDataExchangeReceive.systemFixed.SMES_Active )
      I_Contact( #stateHideAlarm.smesactive )
      { S7_Templates := "time_type := Time" } #instKistlerOnDelay.TON(pt := #cfgKistlerOnDelay, et =>)
      S_Coil( #stateAlarm.smesActive )
   END_RUNG
   RUNG wire#w4
      Contact( #statDataExchangeReceive.systemFixed.SMST2_Active )
      I_Contact( #stateHideAlarm.smst2active )
      S_Coil( #stateAlarm.smst2active )
   END_RUNG
   RUNG wire#w4
      Contact( #statDataExchangeReceive.systemFixed.SMM1_Active )
      I_Contact( #stateHideAlarm.smm1Active )
      S_Coil( #stateAlarm.smm1active )
   END_RUNG
   RUNG wire#w4
      I_Contact( #statDataExchangeReceive.systemFixed.SMES_Active )
      I_Contact( #statDataExchangeReceive.systemFixed.SMST2_Active )
      I_Contact( #statDataExchangeReceive.systemFixed.SMM1_Active )
      wire#w5
      I_Contact( #statDataExchangeReceive.systemFixed.Alarm )
      I_Contact( #statDataExchangeReceive.systemFixed.ServoError )
      Contact( #statDataExchangeSend.systemFixed.DriveEnable )
      I_Contact( #statDataExchangeReceive.systemFixed.DriveEnabled )
      I_Contact( #servoNotInstalled )
      { S7_Templates := "time_type := Time" } #statInstruction.driveEnableTMR.TON(pt := T#0.6s, et =>)
      S_Coil( #stateAlarm.driveenabledNOK )
   END_RUNG
   RUNG wire#w5
      Contact( #statDataExchangeReceive.systemFixed.Alarm )
      I_Contact( #stateHideAlarm.Alarm )
      S_Coil( #stateAlarm.alarm )
   END_RUNG
   RUNG wire#w4
      Contact( #statDataExchangeSend.systemFixed.DriveEnable )
      wire#w6
      Contact( #strobeEnable )
      Contact( #aux.runSequence )
      Contact( #statDataExchangeReceive.systemFixed.TransmissionFault )
      I_Contact( #stateHideAlarm.transmissionFault )
      S_Coil( #stateAlarm.transmissionFault )
   END_RUNG
   RUNG wire#w6
      Contact( #statDataExchangeSend.systemFixed.RunSequence )
      I_Contact( #continuewait )
      I_Contact( #statDataExchangeReceive.systemFixed.Alarm )
      I_Contact( #statDataExchangeReceive.systemFixed.ServoError )
      P_Trig( #ons[2] )
      Contact( #statDataExchangeReceive.systemFixed.WaitRequest )
      I_Contact( #stateHideAlarm.noContinueWaitCommand )
      S_Coil( #stateAlarm.noContinueWaitCommand )
   END_RUNG
   RUNG wire#w4
      Contact( #aux.automaticMode )
      wire#w7
      Contact( #autoHomePosition )
      wire#w8
      I_Contact( #enablehomePos )
      I_Contact( #stateHideAlarm.enableHomePos )
      S_Coil( #stateAlarm.enableHomePos )
   END_RUNG
   RUNG wire#w4
      Contact( #aux.singleStepMode )
   END_RUNG wire#w7
   RUNG wire#w4
      Contact( #OpModeUserInterfaceOut.opmodeStatus.manualActive )
      Contact( #interfaceHmi[#tecUnitNumber].move.%X2 )
   END_RUNG wire#w8
   RUNG wire#w4
      Contact( #aux.automaticMode )
      wire#w9
      Contact( #autoRunSequence )
      wire#w10
      I_Contact( #enableRunSequence )
      I_Contact( #stateHideAlarm.enableRunSequence )
      S_Coil( #stateAlarm.enableRunSequence )
   END_RUNG
   RUNG wire#w4
      Contact( #aux.singleStepMode )
   END_RUNG wire#w9
   RUNG wire#w4
      Contact( #OpModeUserInterfaceOut.opmodeStatus.manualActive )
      Contact( #interfaceHmi[#tecUnitNumber].move.%X1 )
   END_RUNG wire#w10
   RUNG wire#w1
      I_Contact( #aux.remoteControl )
      Coil( #stateAlarm.remoteControlNotActive )
   END_RUNG
   // the same network as SCL:
   #_w1 := #enableBlock AND NOT #aux.generalAlarm;
   IF #_w1 AND NOT #HardwareOK AND NOT #stateHideAlarm.hardwareNOK THEN
       #stateAlarm.hardwareNOK := TRUE;
   END_IF;
   #_w2 := #_w1 AND #HardwareOK;
   IF #_w2 AND NOT #SafetyOK AND NOT #stateHideAlarm.hardwareNOK THEN #stateAlarm.safetyNOK := TRUE; END_IF;
   #_w3 := #_w2 AND #SafetyOK;
   #instKistlerOnDelay(IN := #_w3 AND #statDataExchangeReceive.systemFixed.SMES_Active AND NOT #stateHideAlarm.smesactive,   // TON
                       PT := #cfgKistlerOnDelay);
   IF #instKistlerOnDelay.Q THEN #stateAlarm.smesActive := TRUE; END_IF;
   IF #_w3 AND #statDataExchangeReceive.systemFixed.SMST2_Active AND NOT #stateHideAlarm.smst2active THEN
       #stateAlarm.smst2active := TRUE;
   END_IF;
   IF #_w3 AND #statDataExchangeReceive.systemFixed.SMM1_Active AND NOT #stateHideAlarm.smm1Active THEN
       #stateAlarm.smm1active := TRUE;
   END_IF;
   #_w4 := #_w3 AND NOT #statDataExchangeReceive.systemFixed.SMES_Active AND NOT #statDataExchangeReceive.systemFixed.SMST2_Active AND NOT #statDataExchangeReceive.systemFixed.SMM1_Active;
   #statInstruction.driveEnableTMR.TON(IN := #_w4 AND NOT #statDataExchangeReceive.systemFixed.Alarm AND NOT #statDataExchangeReceive.systemFixed.ServoError AND #statDataExchangeSend.systemFixed.DriveEnable AND NOT #statDataExchangeReceive.systemFixed.DriveEnabled AND NOT #servoNotInstalled,
                           PT := T#0.6s);
   IF #statInstruction.driveEnableTMR.Q THEN #stateAlarm.driveenabledNOK := TRUE; END_IF;
   IF #_w4 AND #statDataExchangeReceive.systemFixed.Alarm AND NOT #stateHideAlarm.Alarm THEN
       #stateAlarm.alarm := TRUE;
   END_IF;
   #_w5 := #_w3 AND #statDataExchangeSend.systemFixed.DriveEnable;
   IF #_w5 AND #strobeEnable AND #aux.runSequence AND #statDataExchangeReceive.systemFixed.TransmissionFault AND NOT #stateHideAlarm.transmissionFault THEN
       #stateAlarm.transmissionFault := TRUE;
   END_IF;
   #_w6 := #_w5 AND #statDataExchangeSend.systemFixed.RunSequence AND NOT #continuewait AND NOT #statDataExchangeReceive.systemFixed.Alarm AND NOT #statDataExchangeReceive.systemFixed.ServoError;
   #_w7 := #_w6 AND NOT #ons[2];   // rising edge
   #ons[2] := #_w6;
   IF #_w7 AND #statDataExchangeReceive.systemFixed.WaitRequest AND NOT #stateHideAlarm.noContinueWaitCommand THEN
       #stateAlarm.noContinueWaitCommand := TRUE;
   END_IF;
   IF #_w3 AND (((#aux.automaticMode OR #aux.singleStepMode) AND #autoHomePosition) OR (#OpModeUserInterfaceOut.opmodeStatus.manualActive AND #interfaceHmi[#tecUnitNumber].move.%X2)) AND NOT #enablehomePos AND NOT #stateHideAlarm.enableHomePos THEN
       #stateAlarm.enableHomePos := TRUE;
   END_IF;
   IF #_w3 AND (((#aux.automaticMode OR #aux.singleStepMode) AND #autoRunSequence) OR (#OpModeUserInterfaceOut.opmodeStatus.manualActive AND #interfaceHmi[#tecUnitNumber].move.%X1)) AND NOT #enableRunSequence AND NOT #stateHideAlarm.enableRunSequence THEN
       #stateAlarm.enableRunSequence := TRUE;
   END_IF;
   #stateAlarm.remoteControlNotActive := #enableBlock AND NOT #aux.remoteControl;
END_REGION

REGION Network 39 (SCL): Evaluate Internal Alarms
   // Processes internal fault conditions: driveenabledNOK, timerMonitorRunSequence, timerMonitorHomePos, timerMonitorReferencePos, noContinueWaitCommand, safetyNOK, smesActive, and serialnumbermismatch. Latches each into stateAlarm bits.
   #statInternalAlarmNoPD := 0;

   FOR #statAlarmByteIndex := 28 TO 35 DO
       #internalFaultCode[(#statAlarmByteIndex - 28) * 8] := #statDataExchangeReceive.userDefinedOutData[#statAlarmByteIndex].%X0;
       #internalFaultCode[(#statAlarmByteIndex - 28) * 8 + 1] := #statDataExchangeReceive.userDefinedOutData[#statAlarmByteIndex].%X1;
       #internalFaultCode[(#statAlarmByteIndex - 28) * 8 + 2] := #statDataExchangeReceive.userDefinedOutData[#statAlarmByteIndex].%X2;
       #internalFaultCode[(#statAlarmByteIndex - 28) * 8 + 3] := #statDataExchangeReceive.userDefinedOutData[#statAlarmByteIndex].%X3;
       #internalFaultCode[(#statAlarmByteIndex - 28) * 8 + 4] := #statDataExchangeReceive.userDefinedOutData[#statAlarmByteIndex].%X4;
       #internalFaultCode[(#statAlarmByteIndex - 28) * 8 + 5] := #statDataExchangeReceive.userDefinedOutData[#statAlarmByteIndex].%X5;
       #internalFaultCode[(#statAlarmByteIndex - 28) * 8 + 6] := #statDataExchangeReceive.userDefinedOutData[#statAlarmByteIndex].%X6;
       #internalFaultCode[(#statAlarmByteIndex - 28) * 8 + 7] := #statDataExchangeReceive.userDefinedOutData[#statAlarmByteIndex].%X7;
   END_FOR;
END_REGION

REGION Network 40: Fault General Alarm
   // OR-combines all active visible alarm bits into the GeneralAlarm output. Also sets aux.generalAlarm. GeneralAlarm TRUE blocks the ready output and drives ProDiag supervision to annunciate the fault.
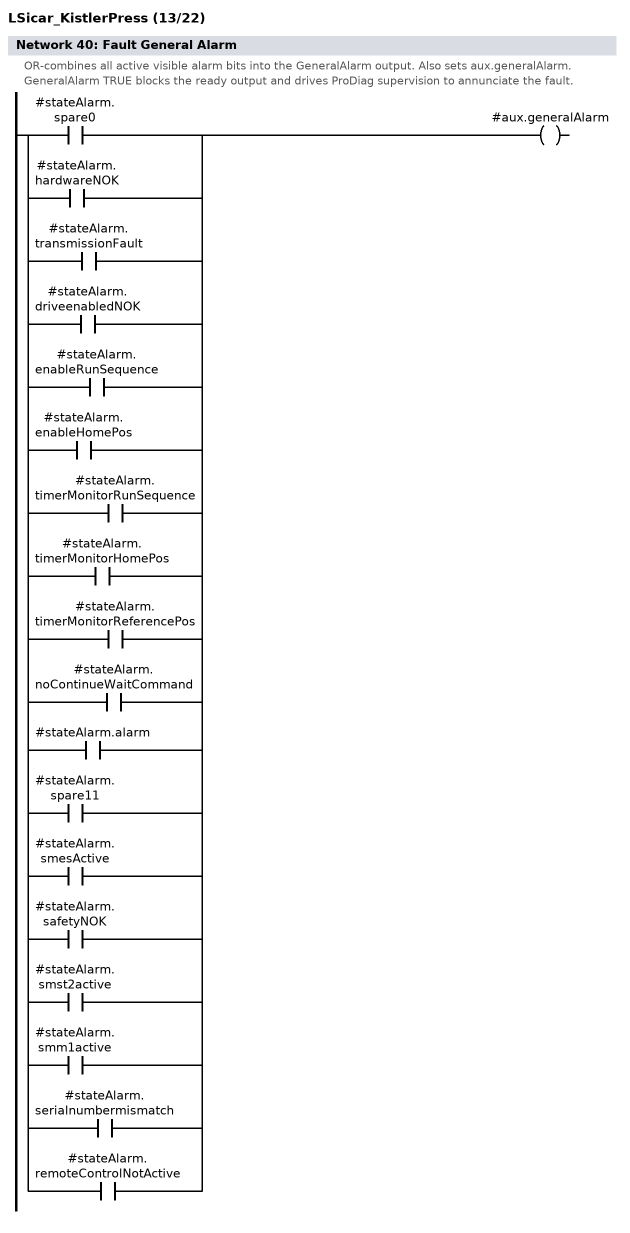
   RUNG wire#powerrail
      Contact( #stateAlarm.spare0 )
      wire#w1
      Coil( #aux.generalAlarm )
   END_RUNG
   RUNG wire#powerrail
      Contact( #stateAlarm.hardwareNOK )
   END_RUNG wire#w1
   RUNG wire#powerrail
      Contact( #stateAlarm.transmissionFault )
   END_RUNG wire#w1
   RUNG wire#powerrail
      Contact( #stateAlarm.driveenabledNOK )
   END_RUNG wire#w1
   RUNG wire#powerrail
      Contact( #stateAlarm.enableRunSequence )
   END_RUNG wire#w1
   RUNG wire#powerrail
      Contact( #stateAlarm.enableHomePos )
   END_RUNG wire#w1
   RUNG wire#powerrail
      Contact( #stateAlarm.timerMonitorRunSequence )
   END_RUNG wire#w1
   RUNG wire#powerrail
      Contact( #stateAlarm.timerMonitorHomePos )
   END_RUNG wire#w1
   RUNG wire#powerrail
      Contact( #stateAlarm.timerMonitorReferencePos )
   END_RUNG wire#w1
   RUNG wire#powerrail
      Contact( #stateAlarm.noContinueWaitCommand )
   END_RUNG wire#w1
   RUNG wire#powerrail
      Contact( #stateAlarm.alarm )
   END_RUNG wire#w1
   RUNG wire#powerrail
      Contact( #stateAlarm.spare11 )
   END_RUNG wire#w1
   RUNG wire#powerrail
      Contact( #stateAlarm.smesActive )
   END_RUNG wire#w1
   RUNG wire#powerrail
      Contact( #stateAlarm.safetyNOK )
   END_RUNG wire#w1
   RUNG wire#powerrail
      Contact( #stateAlarm.smst2active )
   END_RUNG wire#w1
   RUNG wire#powerrail
      Contact( #stateAlarm.smm1active )
   END_RUNG wire#w1
   RUNG wire#powerrail
      Contact( #stateAlarm.serialnumbermismatch )
   END_RUNG wire#w1
   RUNG wire#powerrail
      Contact( #stateAlarm.remoteControlNotActive )
   END_RUNG wire#w1
   // the same network as SCL:
   #aux.generalAlarm := #stateAlarm.spare0 OR #stateAlarm.hardwareNOK OR #stateAlarm.transmissionFault OR #stateAlarm.driveenabledNOK OR #stateAlarm.enableRunSequence OR #stateAlarm.enableHomePos OR #stateAlarm.timerMonitorRunSequence OR #stateAlarm.timerMonitorHomePos OR #stateAlarm.timerMonitorReferencePos OR #stateAlarm.noContinueWaitCommand OR #stateAlarm.alarm OR #stateAlarm.spare11 OR #stateAlarm.smesActive OR #stateAlarm.safetyNOK OR #stateAlarm.smst2active OR #stateAlarm.smm1active OR #stateAlarm.serialnumbermismatch OR #stateAlarm.remoteControlNotActive;
END_REGION

REGION Network 41: Map Alarms to HMI Interface Alarm
   // Writes the active alarm word and individual alarm bit states into the interfaceHmi array elements for HMI alarm display, acknowledgement, and remote reset functionality on the operator panel.
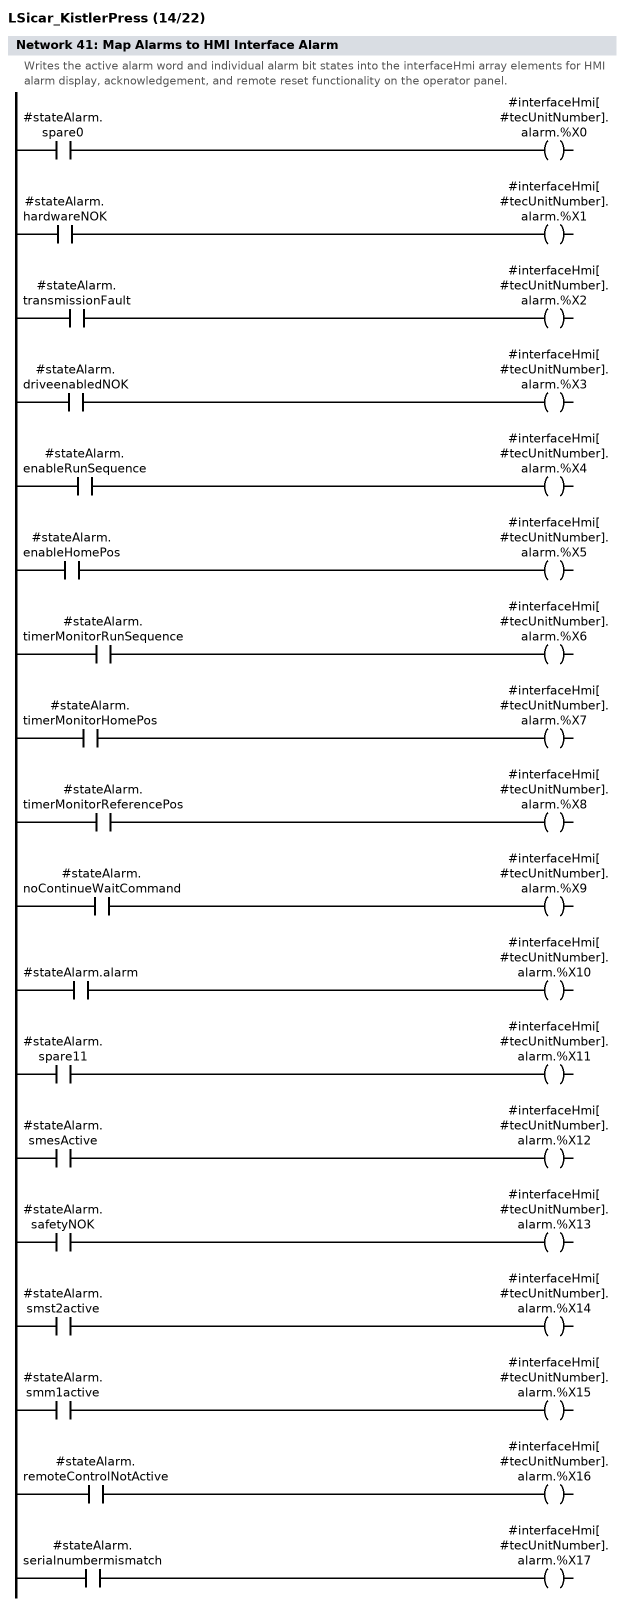
   RUNG wire#powerrail
      Contact( #stateAlarm.spare0 )
      Coil( #interfaceHmi[#tecUnitNumber].alarm.%X0 )
   END_RUNG
   RUNG wire#powerrail
      Contact( #stateAlarm.hardwareNOK )
      Coil( #interfaceHmi[#tecUnitNumber].alarm.%X1 )
   END_RUNG
   RUNG wire#powerrail
      Contact( #stateAlarm.transmissionFault )
      Coil( #interfaceHmi[#tecUnitNumber].alarm.%X2 )
   END_RUNG
   RUNG wire#powerrail
      Contact( #stateAlarm.driveenabledNOK )
      Coil( #interfaceHmi[#tecUnitNumber].alarm.%X3 )
   END_RUNG
   RUNG wire#powerrail
      Contact( #stateAlarm.enableRunSequence )
      Coil( #interfaceHmi[#tecUnitNumber].alarm.%X4 )
   END_RUNG
   RUNG wire#powerrail
      Contact( #stateAlarm.enableHomePos )
      Coil( #interfaceHmi[#tecUnitNumber].alarm.%X5 )
   END_RUNG
   RUNG wire#powerrail
      Contact( #stateAlarm.timerMonitorRunSequence )
      Coil( #interfaceHmi[#tecUnitNumber].alarm.%X6 )
   END_RUNG
   RUNG wire#powerrail
      Contact( #stateAlarm.timerMonitorHomePos )
      Coil( #interfaceHmi[#tecUnitNumber].alarm.%X7 )
   END_RUNG
   RUNG wire#powerrail
      Contact( #stateAlarm.timerMonitorReferencePos )
      Coil( #interfaceHmi[#tecUnitNumber].alarm.%X8 )
   END_RUNG
   RUNG wire#powerrail
      Contact( #stateAlarm.noContinueWaitCommand )
      Coil( #interfaceHmi[#tecUnitNumber].alarm.%X9 )
   END_RUNG
   RUNG wire#powerrail
      Contact( #stateAlarm.alarm )
      Coil( #interfaceHmi[#tecUnitNumber].alarm.%X10 )
   END_RUNG
   RUNG wire#powerrail
      Contact( #stateAlarm.spare11 )
      Coil( #interfaceHmi[#tecUnitNumber].alarm.%X11 )
   END_RUNG
   RUNG wire#powerrail
      Contact( #stateAlarm.smesActive )
      Coil( #interfaceHmi[#tecUnitNumber].alarm.%X12 )
   END_RUNG
   RUNG wire#powerrail
      Contact( #stateAlarm.safetyNOK )
      Coil( #interfaceHmi[#tecUnitNumber].alarm.%X13 )
   END_RUNG
   RUNG wire#powerrail
      Contact( #stateAlarm.smst2active )
      Coil( #interfaceHmi[#tecUnitNumber].alarm.%X14 )
   END_RUNG
   RUNG wire#powerrail
      Contact( #stateAlarm.smm1active )
      Coil( #interfaceHmi[#tecUnitNumber].alarm.%X15 )
   END_RUNG
   RUNG wire#powerrail
      Contact( #stateAlarm.remoteControlNotActive )
      Coil( #interfaceHmi[#tecUnitNumber].alarm.%X16 )
   END_RUNG
   RUNG wire#powerrail
      Contact( #stateAlarm.serialnumbermismatch )
      Coil( #interfaceHmi[#tecUnitNumber].alarm.%X17 )
   END_RUNG
   // the same network as SCL:
   #interfaceHmi[#tecUnitNumber].alarm.%X0 := #stateAlarm.spare0;
   #interfaceHmi[#tecUnitNumber].alarm.%X1 := #stateAlarm.hardwareNOK;
   #interfaceHmi[#tecUnitNumber].alarm.%X2 := #stateAlarm.transmissionFault;
   #interfaceHmi[#tecUnitNumber].alarm.%X3 := #stateAlarm.driveenabledNOK;
   #interfaceHmi[#tecUnitNumber].alarm.%X4 := #stateAlarm.enableRunSequence;
   #interfaceHmi[#tecUnitNumber].alarm.%X5 := #stateAlarm.enableHomePos;
   #interfaceHmi[#tecUnitNumber].alarm.%X6 := #stateAlarm.timerMonitorRunSequence;
   #interfaceHmi[#tecUnitNumber].alarm.%X7 := #stateAlarm.timerMonitorHomePos;
   #interfaceHmi[#tecUnitNumber].alarm.%X8 := #stateAlarm.timerMonitorReferencePos;
   #interfaceHmi[#tecUnitNumber].alarm.%X9 := #stateAlarm.noContinueWaitCommand;
   #interfaceHmi[#tecUnitNumber].alarm.%X10 := #stateAlarm.alarm;
   #interfaceHmi[#tecUnitNumber].alarm.%X11 := #stateAlarm.spare11;
   #interfaceHmi[#tecUnitNumber].alarm.%X12 := #stateAlarm.smesActive;
   #interfaceHmi[#tecUnitNumber].alarm.%X13 := #stateAlarm.safetyNOK;
   #interfaceHmi[#tecUnitNumber].alarm.%X14 := #stateAlarm.smst2active;
   #interfaceHmi[#tecUnitNumber].alarm.%X15 := #stateAlarm.smm1active;
   #interfaceHmi[#tecUnitNumber].alarm.%X16 := #stateAlarm.remoteControlNotActive;
   #interfaceHmi[#tecUnitNumber].alarm.%X17 := #stateAlarm.serialnumbermismatch;
END_REGION

